		(* build template for Outer *)
		fbBuildOACData(
			bExecute		:= TRUE,
			bAddXMLHEader	:= FALSE,
			nTabIndent		:= 1,
			nOuterIndex		:= nOuterIndex,
			stOACData		:= stCACData.Outer[nOuterIndex]
		);

		(* build OAC data complete *)
		IF fbBuildOACData.bDone = TRUE THEN

			(* arrCACImage has room for OAC data and trailing </Case> tag (if required) *)
			IF SIZEOF(arrCACImage) - nCACByte - LEN('</Case>') > fbBuildOACData.nOACByte THEN

				(* add Outer data to arrCACImage *)
				(*MEMMOVE(ADR(arrCACImage[nCACByte]), ADR(fbBuildOACData.arrOACImage), fbBuildOACData.nOACByte);
				nCACByte := nCACByte + fbBuildOACData.nOACByte;*)

				nControlSize := nControlSize + fbBuildOACData.nOACByte;
				IF nControlSize <  nMaxCACImageSize  AND stCACData.NumberOfOuters <> 0 THEN
					MEMMOVE(ADR(arrCACImage[nCACByte]), ADR(fbBuildOACData.arrOACImage), fbBuildOACData.nOACByte);
					nCACByte := nCACByte + fbBuildOACData.nOACByte;
				ELSE
					bBufferOverflow	:=TRUE;
					bDone := TRUE;
					(*RETURN;*)
				END_IF


				(* last Outer in Case *)
				IF nOuterIndex = stCACData.NumberOfOuters OR  stCACData.NumberOfOuters = 0 THEN

					(* append </Case> tag *)
					strString := '</Case>';
					AppendImageData();
				END_IF
			END_IF

			eState := E_CAC_WRITEXMLIMAGE;

			(* close off fbBuildOACData *)
			fbBuildOACData(bExecute := FALSE);
		END_IF

	(* write CAC file template *)
	E_CAC_WRITEXMLIMAGE:

		(* write data to file *)
		fbWriteFile(
			sNetId		:= '',
			hFile		:= hFile,
			pWriteBuff	:= ADR(arrCACImage),
			cbWriteLen	:= nCACByte,
			bExecute	:= TRUE,
			tTimeout	:= T#1s
		);

		(* write file complete *)
		IF fbWriteFile.bBusy = FALSE THEN

			(* write file completed OK *)
			IF fbWriteFile.bError = FALSE THEN

				(* OAC required and more OAC data to be written *)
				IF nOuterIndex < stCACData.NumberOfOuters THEN

					(* re-initialise CAC byte and output image *)
					nCACByte := 0;
					nControlSize := 0;
					MEMSET(ADR(arrCACImage), 16#00, SIZEOF(arrCACImage));
					(* next Outer in Case *)
					nOuterIndex := nOuterIndex + 1;

					eState := E_CAC_BUILDXMLIMAGE;

				(* all Outers added to CAC file or Outer data not required *)
				ELSE
					eState := E_CAC_CLOSEFILE;
				END_IF
			(* write file error *)
			ELSE

				bError := TRUE;
				nErrorID := fbWriteFile.nErrID;
				eErrorState := eState;

				eState := E_CAC_CLOSEFILE;
			END_IF

			(* close off fbWriteFile *)
			fbWriteFile(bExecute := FALSE);
		END_IF


	(* close CAC template *)
	E_CAC_CLOSEFILE:

		(* close file *)
		fbCloseFile(
			sNetId		:= '',
			hFile		:= hFile,
			bExecute	:= TRUE,
			tTimeout	:= T#1s
		);

		(* close file complete *)
		IF fbCloseFile.bBusy = FALSE THEN

			(* close file completed OK and no file write error *)
			IF fbCloseFile.bError = FALSE AND bError = FALSE THEN

				eState := E_CAC_DONE;

			(* close file error or previous error with file write *)
			ELSE

				(* no previous error *)
				IF bError = FALSE THEN

					(* update error status *)
					bError := FALSE;
					nErrorID := fbCloseFile.nErrId;
					eErrorState := eState;
				END_IF

				eState := E_CAC_DONE;
			END_IF

			(* close off fbCloseFile *)
			fbCloseFile(bExecute := FALSE);
		END_IF

	(* complete *)
	E_CAC_DONE:

		bDone := TRUE;
		bBusy := FALSE;

		eState := E_CAC_IDLE;

(* unknown state *)
ELSE

	eState := E_CAC_IDLE;
END_CASE

ACTION AppendImageData:
nStringLen := LEN(strString);
nControlSize := nControlSize + nStringLen;
IF nControlSize <  nMaxCACImageSize THEN
	MEMMOVE(ADR(arrCACImage[nCACByte]), ADR(strString), nStringLen);
	nCACByte := nCACByte + nStringLen;
ELSE
	bBufferOverflow	:=TRUE;
	bDone := TRUE;
	(*RETURN;*)
END_IF
END_ACTION

END_FUNCTION_BLOCK

// ---- POUs/_Exclude/FB_CHM_ClearArchive.TcPOU
(* scans CHM archive and deletes files and folders older than tMaxArchiveAge *)
FUNCTION_BLOCK FB_CHM_ClearArchive
VAR_INPUT
	bExecute				: BOOL;			(* set TRUE to scan archive for old folders and files *)
	tMaxArchiveAge		: TIME;			(* max file age, older files/folders will be deleted *)
	strLocalCHMPath		: STRING(255);	(* CaseTrace CHM folder path *)
	sSystemTime			: TIMESTRUCT;	(* current system time *)
END_VAR
VAR_OUTPUT
	bDone				: BOOL;			(* TRUE = scan complete *)
	bBusy				: BOOL;			(* TRUE = scan in progress *)
	bError				: BOOL;			(* TRUE = scan error *)
	nErrorID				: UDINT;		(* error code *)
	nFoldersDeleted		: UDINT;		(* total folders deleted *)
	nCHMFilesDeleted		: UDINT;		(* total CHM files deleted *)
END_VAR
VAR
	fbExecute				: R_TRIG;
	eState				: E_CHM_State;
	eErrorState			: E_CHM_State;
	nSourceAge			: T_ULARGE_INTEGER;
	nFoldersFound			: UDINT;
	nCHMFilesFound		: UDINT;

	fbFindFolder			: FB_EnumFindFileEntry;
	eFolderCmd 			: E_EnumCmdType := eEnumCmd_First;
	strFolder				: STRING(255);

	fbFindFile				: FB_EnumFindFileEntry;
	eFileCmd 				: E_EnumCmdType := eEnumCmd_First;
	strFileName			: STRING(255);

	fbDeleteFile			: FB_FileDelete;
	fbDeleteFolder			: FB_RemoveDir;
END_VAR

fbExecute(CLK := bExecute);

CASE eState OF

	(* idle *)
	E_CHM_IDLE:

		(* rising edge of bExecute *)
		IF fbExecute.Q = TRUE THEN

			(* update outputs *)
			bDone := FALSE;
			bBusy := TRUE;
			bError := FALSE;
			nErrorID := 0;

			(* reset values *)
			nFoldersDeleted := 0;
			nCHMFilesDeleted := 0;
			nFoldersFound := 0;
			nCHMFilesFound := 0;

			strFolder := '';
			eFolderCmd := eEnumCmd_First;
			strFileName := '';
			eFileCmd := eEnumCmd_First;

			eState := E_CHM_FINDFOLDER;

		(* bExecute has been reset *)
		ELSIF bExecute = FALSE THEN

			(* reset outputs *)
			bDone := FALSE;
			bBusy := FALSE;
			bError := FALSE;
			nErrorID := 0;
		END_IF


	(* date folders *)
	E_CHM_FINDFOLDER:

		(* get list of date folders in "..CaseTrace\CHM\Archive\" *)
		fbFindFolder(
			sNetId		:= '',
			sPathName	:= CONCAT(strLocalCHMPath, 'Archive\*.'),
			eCmd		:= eFolderCmd,
			bExecute	:= TRUE,
			tTimeout	:= T#5s
		);

		(* find folder complete *)
		IF fbFindFolder.bBusy = FALSE THEN

			(* find folder completed OK *)
			IF fbFindFolder.bError = FALSE THEN

				(* file list complete *)
				IF fbFindFolder.bEOE = TRUE THEN

					eFolderCmd := eEnumCmd_First;

					eState := E_CHM_DONE;

				(* file found *)
				ELSE

					(* first 2 folders are '.' and '..' *)
					IF fbFindFolder.stFindFile.sFileName = '.' OR fbFindFolder.stFindFile.sFileName = '..' THEN

						(* next file *)
						eFolderCmd := eEnumCmd_Next;

					(* folder found *)
					ELSE

						(* update counter *)
						nFoldersFound := nFoldersFound + 1;

						(* FolderAge = SystemTime - FileTime *)
						nSourceAge := UInt64Sub64(F_FileTimeToULarge(SYSTEMTIME_TO_FILETIME(sSystemTime)), F_FileTimeToULarge(fbFindFolder.stFindFile.creationTime));

						(* folder is older than max age (converted to 64-bit format) *)
						IF UInt64Cmp64(nSourceAge, UInt32x32To64(TIME_TO_UDINT(tMaxArchiveAge), 10000)) = 1 THEN

							(* folder found *)
							strFolder := fbFindFolder.stFindFile.sFileName;

							eState := E_CHM_FINDFILE;
						END_IF

						(* next folder on next pass *)
						eFolderCmd := eEnumCmd_Next;
					END_IF
				END_IF

			(* find folder error *)
			ELSE

				(* update outputs *)
				bError := TRUE;
				nErrorID := fbFindFolder.nErrID;
				eErrorState := eState;

				eFolderCmd := eEnumCmd_First;

				eState := E_CHM_DONE;
			END_IF

			(* close off fbFindFolder *)
			fbFindFolder(bExecute := FALSE);
		END_IF


	(* find files in folder *)
	E_CHM_FINDFILE:

		(* get list of files *)
		fbFindFile(
			sNetId		:= '',
			sPathName	:= F_CONCAT4(strLocalCHMPath, 'Archive\', strFolder, '\*.*'),
			eCmd		:= eFileCmd,
			bExecute	:= TRUE,
			tTimeout	:= T#5s
		);

		(* find date complete *)
		IF fbFindFile.bBusy = FALSE THEN

			(* find file completed OK *)
			IF fbFindFile.bError = FALSE THEN

				(* file list complete *)
				IF fbFindFile.bEOE = TRUE THEN

					eFileCmd := eEnumCmd_First;

					eState := E_CHM_DELETEFOLDER;

				(* file found *)
				ELSE

					(* first 2 files could be '.' and '..' *)
					IF fbFindFile.stFindFile.sFileName = '.' OR fbFindFile.stFindFile.sFileName = '..' THEN

						(* next file *)
						eFileCmd := eEnumCmd_Next;

					(* folder found *)
					ELSE

						(* count files in folder *)
						nCHMFilesFound := nCHMFilesFound + 1;
	
						(* FileAge = SystemTime - FileTime *)
						nSourceAge := UInt64Sub64(F_FileTimeToULarge(SYSTEMTIME_TO_FILETIME(sSystemTime)), F_FileTimeToULarge(fbFindFile.stFindFile.creationTime));

						(* source file is older than max age (converted to 64-bit format) *)
						IF UInt64Cmp64(nSourceAge, UInt32x32To64(TIME_TO_UDINT(tMaxArchiveAge), 10000)) = 1 THEN
	
							(* date folder found *)
							strFileName := fbFindFile.stFindFile.sFileName;
	
							eState := E_CHM_DELETEFILE;
						END_IF
	
						(* next folder *)
						eFileCmd := eEnumCmd_Next;
					END_IF
				END_IF

			(* find file error *)
			ELSE

				(* update outputs *)
				bError := TRUE;
				nErrorID := fbFindFile.nErrID;
				eErrorState := eState;

				eFileCmd := eEnumCmd_First;

				eState := E_CHM_FINDFOLDER;
			END_IF

			(* close off fbFindFile *)
			fbFindFile(bExecute := FALSE);
		END_IF


	(* delete old file *)
	E_CHM_DELETEFILE:

		(* delete files *)
		fbDeleteFile(
			sNetId		:= '',
			sPathName	:= F_CONCAT5(strLocalCHMPath, 'Archive\', strFolder, '\', strFileName),
			ePath		:= PATH_GENERIC,
			bExecute	:= TRUE,
			tTimeout	:= T#1s
		);

		(* delete file complete *)
		IF fbDeleteFile.bBusy = FALSE THEN

			(* delete file completed OK *)
			IF fbDeleteFile.bError = FALSE THEN

				(* count files deleted from current folder *)
				nCHMFilesDeleted := nCHMFilesDeleted + 1;
			END_IF

			eState := E_CHM_FINDFILE;

			(* close off fbDeleteFile *)
			fbDeleteFile(bExecute := FALSE);
		END_IF


	(* delete old folder *)
	E_CHM_DELETEFOLDER:

		(* delete folder *)
		fbDeleteFolder(
			sNetId		:= '',
			sPathName	:= F_CONCAT3(strLocalCHMPath, 'Archive\', strFolder),
			ePath		:= PATH_GENERIC,
			bExecute	:= TRUE,
			tTimeout	:= T#1s
		);

		(* delete folder complete *)
		IF fbDeleteFolder.bBusy = FALSE THEN

			(* delete folder complete *)
			IF fbDeleteFolder.bError = FALSE THEN

				(* count folder deleted *)
				nFoldersDeleted := nFoldersDeleted + 1;
			END_IF

			eState := E_CHM_FINDFOLDER;

			(* close off fbDeleteFolder *)
			fbDeleteFolder(bExecute := FALSE);
		END_IF


	(* complete *)
	E_CHM_DONE:

		(* update outputs *)
		bBusy := FALSE;
		bDone := TRUE;

		eState := E_CHM_IDLE;


(* unknown state *)
ELSE

	eState := E_CHM_IDLE;

	bDone := FALSE;
	bBusy := FALSE;
	bError := FALSE;
	nErrorID := 0;
END_CASE

END_FUNCTION_BLOCK

// ---- POUs/_Exclude/FB_CX_NVData_NOVRAM_4K.TcPOU
(* stores data in local NOV/DP-RAM device (CX only) *)
FUNCTION_BLOCK FB_CX_NVData_NOVRAM_4K
VAR_INPUT
	bEnable				: BOOL;				(* set TRUE to enable NOVRAM data storage *)
	bExport				: BOOL;				(* set TRUE to export data to XML file, format is compatible with TSM export file *)
	bImport				: BOOL;				(* set TRUE to import data from XML file, format is compatible with TSM export file *)
	pCtrlData			: POINTER TO WORD;	(* pointer to 1st byte of ctrl data to be stored *)
	nCtrlBytes			: UDINT;			(* no of ctrl data bytes to be stored *)
	strTransferPathFile	: T_MaxString;		(* transfer file name for export/import *)
END_VAR
VAR_OUTPUT
	bNVDataInitOK		: BOOL;				(* TRUE = initialisation completed OK *)
	bError				: BOOL;				(* TRUE = initialisation error (device or checksum) *)
	nUpdates			: UDINT;			(* number of NOVRAM writes completed *)
	nDeviceID			: WORD;				(* NOVRAM device ID *)
END_VAR
VAR
	eState				: E_CX_NVDataCtrlState;
	eErrorState			: E_CX_NVDataCtrlState;
	arrInputData		: ARRAY[0..4095] OF BYTE;
	arrOutputData		: ARRAY[0..4095] OF BYTE;

	fbExport			: R_TRIG;
	bExportReq			: BOOL;
	fbImport			: R_TRIG;
	bImportReq			: BOOL;

	fbTaskTime			: FB_SYSTEM_TaskInfo;
	nNVReadBlockSize	: UDINT;
	nNVWriteBlockSize	: UDINT;
	nChecksumBlockSize	: UDINT;
	pNVData				: POINTER TO BYTE;

	fbGetCXPlatform		: FB_CxGetDeviceIdentificationEx;
	nMaxDataBytes		: UDINT;
	fbGetDeviceID		: FB_CX_GetDeviceID;
	fbGetDeviceInfo		: FB_GetDPRAMInfo;
	sDeviceInfo			: ST_NovRamAddrInfo;

	nActiveDataArea		: UINT;
	pChecksum			: POINTER TO WORD;
	nCalcChecksum		: WORD;
	nNVBlockOffset		: UDINT;
	nNVBlockBytes		: UDINT;
	nIndexOffset		: UDINT;
	nIndexBlockBytes	: UDINT;
	fbTransferData		: FB_CX_NVData_Transfer;
END_VAR
(*
-------------------------------------------------------------------------------------------------
Date		Version	Author	Comments
-------------------------------------------------------------------------------------------------
30/01/2015	3.00.00	PB		Initial release

-------------------------------------------------------------------------------------------------

*)

(* rising edge of bExport *)
fbExport(CLK := bExport);
IF fbExport.Q = TRUE THEN

	(* set flag to export data at next opportunity *)
	bExportReq := TRUE;
END_IF

(* rising edge of bImport *)
fbImport(CLK := bImport);
IF fbImport.Q = TRUE THEN

	(* set flag to import data at next opportunity *)
	bImportReq := TRUE;
END_IF


CASE eState OF

	(* IDLE state *)
	E_CX_NVDATA_IDLE:

		(* NOVRAM storage is enabled *)
		IF bEnable = TRUE THEN

			(* get current task time *)
			fbTaskTime();

			(* initialise vars *)
			nActiveDataArea := 0;
			nMaxDataBytes := SIZEOF(arrInputData);
			MEMSET(ADR(sDeviceInfo), 16#00, SIZEOF(sDeviceInfo));

			(* initialise outputs *)
			nUpdates := 0;
			nDeviceID := 0;

			eState := E_CX_NVDATA_PLATFORM;

		(* else *)
		ELSE

			bNVDataInitOK := FALSE;
			bError := FALSE;
		END_IF


	(* find CX type *)
	E_CX_NVDATA_PLATFORM:

		(* get CX platform type *)
		fbGetCXPlatform(
			bExecute	:= TRUE,
			tTimeout	:= T#1s
		);

		(* get CX platform type complete *)
		IF fbGetCXPlatform.bBusy = FALSE THEN

			(* get CX platform type completed OK *)
			IF fbGetCXPlatform.bError = FALSE THEN

				(* Block sizes have been selected to use approx 5% resource in 1ms PLC task on CX1020 and CX2020. *)
				(* Processor resource should be lower on CX1030 and CX2030/CX2040 due to higher processor speed. *)
				(* FB will be adjusted for other platforms when they are available for testing *)

				(* CX1020/CX1030 platform *)
				IF FIND(fbGetCXPlatform.stDevIdent.strHardwareModel, '1020') > 0 OR FIND(fbGetCXPlatform.stDevIdent.strHardwareModel, '1030') > 0 THEN

					(* NOVRAM block access size per 1ms of PLC cycle time:  READ = 32 bytes/ms, WRITE = 128 bytes/ms *)
					nNVReadBlockSize := MIN(LREAL_TO_UDINT(fbTaskTime.fTaskTimeMicrosecs * 32.0 / 1000.0), 32);
					nNVWriteBlockSize := MIN(LREAL_TO_UDINT(fbTaskTime.fTaskTimeMicrosecs * 128.0 / 1000.0), 128);

					(* checksum block size:  512 bytes/ms PLC task time *)
					nChecksumBlockSize := LREAL_TO_UDINT(fbTaskTime.fTaskTimeMicrosecs * 512.0 / 1000.0);

				(* CX2020/CX2030/CX2040 platform *)
				ELSIF FIND(fbGetCXPlatform.stDevIdent.strHardwareModel, '2020') > 0 OR FIND(fbGetCXPlatform.stDevIdent.strHardwareModel, '2030') > 0 OR FIND(fbGetCXPlatform.stDevIdent.strHardwareModel, '2040') > 0 THEN

					(* NOVRAM block access size per 1ms of PLC cycle time:  READ = 64 bytes/ms, WRITE = 1024 bytes/ms *)
					nNVReadBlockSize := MIN(LREAL_TO_UINT(fbTaskTime.fTaskTimeMicrosecs * 64.0 / 1000.0), 64);
					nNVWriteBlockSize := MIN(LREAL_TO_UINT(fbTaskTime.fTaskTimeMicrosecs * 1024.0 / 1000.0), 1024);

					(* checksum block size per 1ms of PLC cycle time:  1024 bytes/ms *)
					nChecksumBlockSize := LREAL_TO_UINT(fbTaskTime.fTaskTimeMicrosecs * 1024.0 / 1000.0);

				(* CX2020/CX2030/CX2040 platform *)
				ELSIF FIND(fbGetCXPlatform.stDevIdent.strTargetType, 'PC') > 0  THEN

					(* NOVRAM block access size per 1ms of PLC cycle time:  READ = 64 bytes/ms, WRITE = 1024 bytes/ms *)
					nNVReadBlockSize := MIN(LREAL_TO_UINT(fbTaskTime.fTaskTimeMicrosecs * 64.0 / 1000.0), 64);
					nNVWriteBlockSize := MIN(LREAL_TO_UINT(fbTaskTime.fTaskTimeMicrosecs * 1024.0 / 1000.0), 1024);

					(* checksum block size per 1ms of PLC cycle time:  1024 bytes/ms *)
					nChecksumBlockSize := LREAL_TO_UINT(fbTaskTime.fTaskTimeMicrosecs * 1024.0 / 1000.0);
				END_IF

				(* DeviceID is not specified *)
				IF nDeviceID = 0 THEN

					(* search CX for NOVRAM device *)
					eState := E_CX_NVDATA_DEVICEID;

				(* DeviceID is specifeid *)
				ELSE

					(* use specified DeviceID *)
					eState := E_CX_NVDATA_DEVICEINFO;
				END_IF

			(* get CX platform type error *)
			ELSE

				bError := TRUE;
				eErrorState := eState;

				eState := E_CX_NVDATA_DONE;
			END_IF

			(* cloes off fbGetCXPlatform *)
			fbGetCXPlatform(bExecute := FALSE);
		END_IF


	(* find NOVRAM device ID *)
	E_CX_NVDATA_DEVICEID:

		(* get DeviceID for DPRAM *)
		fbGetDeviceID(
			bExecute	:= TRUE,
			eDeviceType	:= IODEVICETYPE_DPRAM
		);

		(* get DeviceID complete *)
		IF fbGetDeviceID.bDone = TRUE THEN

			(* get DeviceID completed OK and NOVRAM device found *)
			IF fbGetDeviceID.bDone = TRUE AND fbGetDeviceID.bDeviceFound = TRUE THEN

				(* DeviceID of NOVRAM device *)
				nDeviceID := fbGetDeviceID.nDeviceID;

				eState := E_CX_NVDATA_DEVICEINFO;

			(* fbGetDeviceID error of NOVRAM device not found *)
			ELSE

				(* reset nDeviceID *)
				nDeviceID := 0;

				(* update error status *)
				bError := TRUE;
				eErrorState := eState;

				eState := E_CX_NVDATA_DONE;
			END_IF

			(* close off fbGetDeviceID *)
			fbGetDeviceID(bExecute := FALSE);
		END_IF


	(* read info of NOVRAM device *)
	E_CX_NVDATA_DEVICEINFO:

		(* get device info *)
		fbGetDeviceInfo(
			nDevId	:= nDeviceID,
			bExecute:= TRUE,
			tTimeOut:= T#1s
		);

		(* device info read complete *)
		IF fbGetDeviceInfo.bBusy = FALSE THEN

			(* NOVRAM info read successful *)
			IF fbGetDeviceInfo.bError = FALSE THEN

				(* set up config data for NV data block *)
				sDeviceInfo := fbGetDeviceInfo.stInfo;

				(* maximum number of NV bytes that can be handled *)
				nMaxDataBytes := sDeviceInfo.iCardMemSize / 2;

				(* specified number of data bytes is valid *)
				IF nCtrlBytes <= nMaxDataBytes THEN

					(* read primary data from NOVRAM *)
					nActiveDataArea := 1;
					pNVData := sDeviceInfo.pCardAddress;

					(* initial byte offset and block size for 1st scan *)
					nNVBlockOffset := 0;
					nNVBlockBytes := MIN(nNVReadBlockSize, nCtrlBytes - nNVBlockOffset);

					eState := E_CX_NVDATA_READ;

				(* memory area too large *)
				ELSE

					bError := TRUE;
					eErrorState := eState;
	
					eState := E_CX_NVDATA_DONE;
				END_IF

			(* unable to read NOVRAM info *)
			ELSE

				bError := TRUE;
				eErrorState := eState;

				eState := E_CX_NVDATA_DONE;
			END_IF

			(* close fbGetDeviceInfo *)
			fbGetDeviceInfo(bExecute:= FALSE);
		END_IF


	(* read data to NOVRAM *)
	E_CX_NVDATA_READ:

		(* restore NOVRAM data into arrInputData in blocks *)
		MEMMOVE(ADR(arrInputData[nNVBlockOffset]), F_PointerToByteADD(pNVData, nNVBlockOffset), nNVBlockBytes);

		(* update memory offset values *)
		nNVBlockOffset := nNVBlockOffset + nNVBlockBytes;
		nNVBlockBytes := MIN(nNVReadBlockSize, nCtrlBytes - nNVBlockOffset);

		(* all bytes transferred *)
		IF nNVBlockOffset >= nCtrlBytes THEN

			(* initialise checksum block vars *)
			nIndexOffset := 0;
			nIndexBlockBytes := MIN(nChecksumBlockSize, nCtrlBytes - 2 - nIndexOffset);
			nCalcChecksum := 16#FFFF;

			eState := E_CX_NVDATA_VALIDATE;
		END_IF


	(* verify checksum *)
	E_CX_NVDATA_VALIDATE:

		(* calculate checksum on block of data *)
		nCalcChecksum := F_DATA_TO_CRC16_CCITT(ADR(arrInputData[nIndexOffset]), nIndexBlockBytes, nCalcChecksum);

		(* update nIndexOffset and nIndexBlockBytes for next pass *)
		nIndexOffset := nIndexOffset + nIndexBlockBytes;
		nIndexBlockBytes := MIN(nChecksumBlockSize, nCtrlBytes - 2 - nIndexOffset);

		(* checksum completed for all bytes *)
		IF nIndexOffset >= nCtrlBytes - 2 THEN

			(* pointer to restored checksum in arrInputData *)
			pChecksum := ADR(arrInputData[nCtrlBytes - 2]);

			(* calculated checksum = restored checksum *)
			IF nCalcChecksum = pChecksum^ THEN

				(* restore NOVRAM data into snapshot array *)
				MEMMOVE(pCtrlData, ADR(arrInputData), nCtrlBytes);
				bNVDataInitOK := TRUE;

				eState := E_CX_NVDATA_COMPARE;

			(* calculated checksum <> restored checksum *)
			ELSE

				(* primary data failed *)
				IF nActiveDataArea = 1 THEN

					(* move to secondary data *)
					nActiveDataArea := 2;

					(* calculate pointers needed to restore secondary data *)
					pNVData := F_PointerToByteADD(pNVData, sDeviceInfo.iCardMemSize / 2);

					(* initial byte offset and block size for 1st scan *)
					nNVBlockOffset := 0;
					nNVBlockBytes := MIN(nNVWriteBlockSize, nCtrlBytes - nNVBlockOffset);

					eState := E_CX_NVDATA_READ;

				(* secondary data failed *)
				ELSE

					(* checksum invalid for primary and secondary data, clear arrInput data *)
					MEMSET(ADR(arrInputData), 16#00, SIZEOF(arrInputData));
					bError := TRUE;
					eErrorState := eState;
					(* data will be written to NOVRAM on COMPARE cycle, unless all values are 0 when no update will occur *)

					eState := E_CX_NVDATA_COMPARE;
				END_IF
			END_IF
		END_IF


	(* snapshot data *)
	E_CX_NVDATA_COMPARE:

		(* FB is enabled *)
		IF bEnable = TRUE THEN

			(* specified number of data bytes is valid *)
			IF nCtrlBytes <= nMaxDataBytes THEN

				(* export data requested *)
				IF bExportReq = TRUE THEN

					(* cancel export flag *)
					bExportReq := FALSE;

					eState := E_CX_NVDATA_EXPORT;

				(* import data requested *)
				ELSIF bImportReq = TRUE THEN

					(* cancel import flag *)
					bImportReq := FALSE;

					eState := E_CX_NVDATA_IMPORT;

				(* check for change of data *)
				ELSE

					(* snapshot data into arrOutputData *)
					MEMMOVE(ADR(arrOutputData), pCtrlData, nCtrlBytes - 2);

					(* snapshot data block does not match terminal data block *)
					IF MEMCMP(ADR(arrOutputData), ADR(arrInputData), nCtrlBytes - 2) <> 0 THEN

						(* initialise checksum block vars *)
						nIndexOffset := 0;
						nIndexBlockBytes := MIN(nChecksumBlockSize, nCtrlBytes - 2 - nIndexOffset);
						nCalcChecksum := 16#FFFF;

						eState := E_CX_NVDATA_CHECKSUM;
					END_IF
				END_IF

			(* memory area too large *)
			ELSE

				bError := TRUE;
				eErrorState := eState;

				eState := E_CX_NVDATA_DONE;
			END_IF

		(* FB is disabled *)
		ELSE

			eState := E_CX_NVDATA_DONE;
		END_IF


	(* calculate checksum for output data *)
	E_CX_NVDATA_CHECKSUM:

		(* calculate checksum on block of data *)
		nCalcChecksum := F_DATA_TO_CRC16_CCITT(ADR(arrOutputData[nIndexOffset]), nIndexBlockBytes, nCalcChecksum);

		(* update nIndexOffset and nIndexBlockBytes for next pass *)
		nIndexOffset := nIndexOffset + nIndexBlockBytes;
		nIndexBlockBytes := MIN(nChecksumBlockSize, nCtrlBytes - 2 - nIndexOffset);

		(* checksum completed for all bytes *)
		IF nIndexOffset >= nCtrlBytes - 2 THEN

			(* pointer to restored checksum in arrInputData *)
			pChecksum := ADR(arrOutputData[nCtrlBytes - 2]);
			pChecksum^ := nCalcChecksum;

			(* write primary data from NOVRAM *)
			nActiveDataArea := 1;
			pNVData := sDeviceInfo.pCardAddress;

			(* initial byte offset and block size for 1st scan *)
			nNVBlockOffset := 0;
			nNVBlockBytes := MIN(nNVWriteBlockSize, nCtrlBytes - nNVBlockOffset);

			eState := E_CX_NVDATA_WRITE;
		END_IF


	(* write data *)
	E_CX_NVDATA_WRITE:

		(* move arrOutputData to NOVRAM *)
		MEMMOVE(F_PointerToByteADD(pNVData, nNVBlockOffset), ADR(arrOutputData[nNVBlockOffset]), nNVBlockBytes);

		(* update memory offset values *)
		nNVBlockOffset := nNVBlockOffset + nNVBlockBytes;
		nNVBlockBytes := MIN(nNVWriteBlockSize, nCtrlBytes - nNVBlockOffset);

		(* all bytes transferred *)
		IF nNVBlockOffset >= nCtrlBytes THEN

			(* primary data written *)
			IF nActiveDataArea = 1 THEN

				(* write primary data from NOVRAM *)
				nActiveDataArea := 2;
				pNVData := F_PointerToByteADD(sDeviceInfo.pCardAddress, sDeviceInfo.iCardMemSize / 2);

				(* initial byte offset and block size for 1st scan *)
				nNVBlockOffset := 0;
				nNVBlockBytes := MIN(nNVWriteBlockSize, nCtrlBytes - nNVBlockOffset);

			(* secondary data complete *)
			ELSE

				(* update outputs *)
				bNVDataInitOK := TRUE;
				bError := FALSE;
				nActiveDataArea := 0;
				nUpdates := nUpdates + 1;

				(* copy arrOutputData to arrInputData *)
				MEMMOVE(ADR(arrInputData), ADR(arrOutputData), nCtrlBytes);

				(* update checksum in pCtrlData area *)
				pChecksum := F_PointerToWordADD(pCtrlData, nCtrlBytes - 2);
				pChecksum^ := nCalcChecksum;

				eState := E_CX_NVDATA_COMPARE;
			END_IF
		END_IF


	(* export data to XML file *)
	E_CX_NVDATA_EXPORT:

		(* export data from arrInputData to XML file *)
		fbTransferData(
			bExecute		:= TRUE,
			bImport			:= FALSE,
			nMaxBlockSize	:= nChecksumBlockSize / 2,
			pCtrlData		:= ADR(arrInputData),
			nCtrlBytes		:= nCtrlBytes,
			strPathFile		:= strTransferPathFile
		);

		(* export data complete *)
		IF fbTransferData.bDone = TRUE THEN

			eState := E_CX_NVDATA_COMPARE;

			(* close off fbTransferData *)
			fbTransferData(bExecute := FALSE);
		END_IF


	(* import data to XML file *)
	E_CX_NVDATA_IMPORT:

		(* import data from XML file to arrOutputData *)
		fbTransferData(
			bExecute		:= TRUE,
			bImport			:= TRUE,
			nMaxBlockSize	:= nChecksumBlockSize / 2,
			pCtrlData		:= ADR(arrOutputData),
			nCtrlBytes		:= SIZEOF(arrOutputData),
			strPathFile		:= strTransferPathFile
		);

		(* import data complete *)
		IF fbTransferData.bDone = TRUE THEN

			(* import data completed OK *)
			IF fbTransferData.bError = FALSE THEN

				(* move data loaded to pCtrlData *)
				MEMMOVE(pCtrlData, ADR(arrOutputData), fbTransferData.nTotalDataBytes);

				eState := E_CX_NVDATA_COMPARE;

			(* import data error *)
			ELSE

				eState := E_CX_NVDATA_COMPARE;
			END_IF

			(* close off fbTransferData *)
			fbTransferData(bExecute := FALSE);
		END_IF


	(* access complete *)
	E_CX_NVDATA_DONE:

		;

END_CASE

END_FUNCTION_BLOCK

// ---- POUs/_Exclude/FB_MemoryMonitor_32K.TcPOU
(* monitor memory area for change of data, max 64Kbytes *)
FUNCTION_BLOCK FB_MemoryMonitor_32K
VAR_INPUT
	bEnable			: BOOL;		(* set TRUE to enable monitoring *)
	pSourceData		: POINTER TO BYTE;	(* pointer to source data *)
	nSourceBytes	: UDINT;	(* no of data bytes *)
	tUpdateTime		: TIME;		(* update time *)
END_VAR
VAR_OUTPUT
	bDataChanged	: BOOL;		(* TRUE = data changed *)
	nTotalChanges	: UDINT;	(* total number of memory changes detected *)
END_VAR
VAR
	arrData			: ARRAY[0..32767] OF BYTE;
	fbUpdateTimer	: FB_PulseGenerator;
END_VAR
(*
-------------------------------------------------------------------------------------------------
Date		Version	Author	Comments
-------------------------------------------------------------------------------------------------
30/01/2015	3.00.00	PB		Initial release

-------------------------------------------------------------------------------------------------
*)

(* update timer *)
fbUpdateTimer(
	bEnable		:= bEnable,
	tPeriod		:= tUpdateTime
);

(* data not changed on last pass *)
IF bDataChanged = FALSE THEN

	(* check for change of data *)
	IF fbUpdateTimer.bOutput = TRUE THEN

		(* source data in array has changed *)
		IF MEMCMP(pSourceData, ADR(arrData), nSourceBytes) <> 0 THEN

			nTotalChanges := nTotalChanges + 1;
			bDataChanged := TRUE;
		END_IF
	END_IF

(* data change detected on last pass *)
ELSE

	(* move data from source to target *)
	MEMMOVE(ADR(arrData), pSourceData, nSourceBytes);
	bDataChanged := FALSE;
END_IF

END_FUNCTION_BLOCK

// ---- POUs/_Exclude/FB_MemoryMonitor_4K.TcPOU
(* monitor memory area for change of data, max 4Kbytes *)
FUNCTION_BLOCK FB_MemoryMonitor_4K
VAR_INPUT
	bEnable			: BOOL;		(* set TRUE to enable monitoring *)
	pSourceData		: POINTER TO BYTE;	(* pointer to source data *)
	nSourceBytes	: UDINT;	(* no of data bytes *)
	tUpdateTime		: TIME;		(* update time *)
END_VAR
VAR_OUTPUT
	bDataChanged	: BOOL;		(* TRUE = data changed *)
	nTotalChanges	: UDINT;	(* total number of memory changes detected *)
END_VAR
VAR
	arrData			: ARRAY[0..4095] OF BYTE;
	fbUpdateTimer	: FB_PulseGenerator;
END_VAR
(*
-------------------------------------------------------------------------------------------------
Date		Version	Author	Comments
-------------------------------------------------------------------------------------------------
30/01/2015	3.00.00	PB		Initial release

-------------------------------------------------------------------------------------------------
*)

(* update timer *)
fbUpdateTimer(
	bEnable		:= bEnable,
	tPeriod		:= tUpdateTime
);

(* data not changed on last pass *)
IF bDataChanged = FALSE THEN

	(* check for change of data *)
	IF fbUpdateTimer.bOutput = TRUE THEN

		(* source data in array has changed *)
		IF MEMCMP(pSourceData, ADR(arrData), nSourceBytes) <> 0 THEN

			nTotalChanges := nTotalChanges + 1;
			bDataChanged := TRUE;
		END_IF
	END_IF

(* data change detected on last pass *)
ELSE

	(* move data from source to target *)
	MEMMOVE(ADR(arrData), pSourceData, nSourceBytes);
	bDataChanged := FALSE;
END_IF

END_FUNCTION_BLOCK

// ---- POUs/_Exclude/FB_OUTER_CompleteDataFromConfirmation.TcPOU
 FUNCTION_BLOCK FB_OUTER_CompleteDataFromConfirmation
VAR_INPUT
	bExecute								: BOOL;		(* set TRUE to scan arrOuterStatus for completed Outers *)
	bValidationTimeout					: BOOL;
	(*bOuterCameraDone					: BOOL;*)
	(*bConfirmationCameraDone			: BOOL;*)
(*	stOuterValidationCameraLastCodes	: ST_SCANNER_ImageData;*)
	stBarcodeConfirmationCameraLastCodes	: ST_SCANNER_ImageData;
	(*nPackPos1								: INT 	:=1;
	nPackPos2								: INT	:=2;*)
	bUseInterimCodeForValidation		: BOOL;
	sLocalOCVPath							: STRING(255);
	stCTDateTime							: ST_SYSTEM_DateTime;	(* CaseTrace date/time structure *)
	bQAReject								: BOOL;
END_VAR
VAR_IN_OUT
	stProductInstruction		: ST_PCM_Status;					(* Product Instruction *)
	stOuterRejectReasons		: ST_RejectReasonsForOuter;
	aOuterStatus				: ARRAY[1..cMAX_OUTER_STATUS_QUEUE] OF ST_OUTER_Status;	(* Outer status register *)
	aOCVPackStatus			: ARRAY[1..cMAX_OUTER_STATUS_QUEUE] OF ST_OUTER_Status;	(* Outer status register *)
	stOuterStatusHMI			: ST_HMI_OuterStatus;
END_VAR
VAR_OUTPUT
	bDone						: BOOL;			(* TRUE = validation complete *)
	bBusy						: BOOL;			(* TRUE = validation in progress *)

	stLastOuterStatus			: ST_OUTER_Status;

	sLastReadOuterBarcode	: T_OUTER_Barcode;
	sLastReadConfPackCode1	: T_PACK_Barcode;
	(*sLastReadConfPackCode2 	: T_PACK_Barcode;*)
	(*aConfPackCodeInPosition		: ARRAY[0..1] OF T_PACK_Barcode;*)
	sOCVRejectCode			: T_RejectCode;
	nOCVRejectID				: UINT;
	bPackDataFoundInStruct	: BOOL;
	nInhibitOCVRestore		: BOOL;
	bReadyToOCVResotre		: BOOL;
	nOutersCompleted			: UDINT;

END_VAR
VAR
	eState						: E_OUTER_AgrregationState;
	fbExecute					: R_TRIG;
	fbTimeOut					: R_TRIG;
	stSystemTime				: TIMESTRUCT;

	(*nAggregartionPackCode	: INT;*)

	nOuterIndex				: INT;
	(*nMaxOuterIndex				: INT;*)
	nPackIndex				: INT;

	aOCVFileCodeName		: ARRAY[1..2] OF T_MaxString;
	bReffedOCVExec			: BOOL;
	fbOCVRefeed				: FB_OUTER_RefeedOCVFilesWtihError; (*FB_PACK_RefeedOCVFilesWtihError;*)

	stPacksDataFromOCV1	: ST_OUTER_Status;
	stPacksDataFromOCV2	: ST_OUTER_Status;

	nTrigID						: UDINT;
	(*aLogTrigID					: ARRAY[0..5] OF UDINT;*)
	nNewOuterTrigID			: UDINT;

	(*aPackStatusValue				: ARRAY[0..10] OF INT;
	aRejectCodePointer            		: ARRAY[0..10] OF STRING(10);

	fbValidatePack					: FB_CODE_ValidateExplicitCode;*)

	nErrorCounter1			: INT;
	nErrorCounter2			: INT;
	nErrorCounter3			: INT;

	tonTestTimer				: TON;
	aLogTimer 					: ARRAY[0..100] OF TIME;
END_VAR

fbExecute(CLK := bExecute);
fbTimeOut(CLK := bValidationTimeout);

stSystemTime := stCTDateTime.sSystemTime;

tonTestTimer(In:= bBusy AND NOT bDone, PT:= t#5000ms);
IF fbTimeOut.Q THEN

		aOuterStatus[1].stOACData.ProductionDate := F_StringWildcard('#YYYYMMDD#', stSystemTime);
		aOuterStatus[1].stOACData.ProductionTime := F_StringWildcard('#hhmmss#', stSystemTime);
		aOuterStatus[1].stOACData.ProductionTimeOffset := F_SYSTEM_SystemTimeOffsetToHHMM(stCTDateTime.nSystemTimeOffset);

		aOuterStatus[1].stOACData.OuterTimeStamp :=F_SYSTEM_SystemTimeAsISO8601(stCTDateTime.sSystemTime, stCTDateTime.sUTCTimeZoneOffset );
		aOuterStatus[1].stOACData.RetailSKU := stProductInstruction.sRetailSKU;
		aOuterStatus[1].stOACData.OuterMachine.ProductionSite :=  stProductInstruction.sProductionSite;
		aOuterStatus[1].stOACData.OuterMachine.ProductionLine := stProductInstruction.sProductionLine;
		aOuterStatus[1].stOACData.BatchNumber := stProductInstruction.sBatchNumber;
		aOuterStatus[1].stOACData.CodingAndTrackingMode := stProductInstruction.nOpMode;

		aOuterStatus[1].stOACData.AcceptanceLevel := stProductInstruction.nAcceptanceLevel;
		aOuterStatus[1].stOACData.NumberOfPacks	:= stProductInstruction.nPacksPerOuter;

		(*IF  NOT bConfirmationCameraDone	THEN
			aOuterStatus[1].sDataSourceTracker	:= 'T_OUT_PCC';
		ELSE
			aOuterStatus[1].sDataSourceTracker	:= 'T_OUT_FB';
		END_IF*)
		aOuterStatus[1].sDataSourceTracker	:= 'T_OUT_FB';

		aOuterStatus[1].nStatus.9 := TRUE;
		aOuterStatus[1].nTriggerID := nNewOuterTrigID;
		aOuterStatus[1].stOACData.OuterRejectCode := stOuterRejectReasons.stOuterTimeOutValidation.sMetsDisplayCode;
		aOuterStatus[1].stOACData.OuterRejectID := stOuterRejectReasons.stOuterTimeOutValidation.nRejectID;

		eState := E_OUTER_DONE_OCV;
END_IF

(* rising edge of bExecute *)
CASE eState OF

	(* idle *)
	E_OUTER_IDLE_OCV:

		(* scan for completed Outer when OAC files are required *)
		IF fbExecute.Q = TRUE THEN

			bDone := FALSE;
			bBusy := TRUE;

			bReffedOCVExec 			:=FALSE;
			bPackDataFoundInStruct 	:=FALSE;
			sOCVRejectCode 			:= '';

			nTrigID					:= 0;
			nNewOuterTrigID := nNewOuterTrigID +1;
			(*MEMMOVE(ADR(aLogTrigID[1]), ADR(aLogTrigID[0]), SIZEOF(aLogTrigID) - SIZEOF(aLogTrigID[0]));*)

			MEMSET(ADR(aOuterStatus[1]), 16#00, SIZEOF(aOuterStatus[1]));
			MEMSET(ADR(stLastOuterStatus), 16#00, SIZEOF(stLastOuterStatus));

			sLastReadOuterBarcode :=  '';
			sLastReadConfPackCode1 :=  '' ;

			MEMSET(ADR(stPacksDataFromOCV1), 16#00, SIZEOF(stPacksDataFromOCV1));
			MEMSET(ADR(stPacksDataFromOCV2), 16#00, SIZEOF(stPacksDataFromOCV2));

			eState := E_OUTER_READ_OCV;

		ELSIF bExecute = FALSE THEN

			(* reset outputs *)
			bDone := FALSE;
			bBusy := FALSE;
		END_IF

	E_OUTER_READ_OCV:

		IF	stProductInstruction.bEnablePacks  THEN

			IF  stBarcodeConfirmationCameraLastCodes.aCodeData[1].strDataString <> ''  THEN

				IF NOT bReffedOCVExec THEN
					FOR nOuterIndex := 1 TO cMAX_OUTER_STATUS_QUEUE  DO

						IF aOCVPackStatus[nOuterIndex].stOACData.AggregationCodes[1] <> '' AND
							aOCVPackStatus[nOuterIndex].stOACData.AggregationCodes[1]   = stBarcodeConfirmationCameraLastCodes.aCodeData[1].strDataString  THEN

							IF NOT  aOCVPackStatus[nOuterIndex].nStatus.22 THEN
								aOuterStatus[1]	 := aOCVPackStatus[nOuterIndex];
								aOuterStatus[1].sDataSourceTracker	:= 'OCV1_AGG';
							ELSE
								aOuterStatus[1].sDataSourceTracker	:= 'BIT22_AGG';
							END_IF
							bPackDataFoundInStruct :=TRUE;
							EXIT;
						END_IF

					END_FOR
				END_IF

				IF bPackDataFoundInStruct AND nOuterIndex > 1 THEN
					nInhibitOCVRestore 			:=FALSE;

					FOR nPackIndex := 1 TO  aOCVPackStatus[nOuterIndex-1].stOACData.NumberOfPacks  DO
							IF aOCVPackStatus[nOuterIndex-1].aOACPackStatus[nPackIndex] <> 5  THEN
									nInhibitOCVRestore :=TRUE;
							END_IF
					END_FOR
				END_IF

				IF NOT bPackDataFoundInStruct  THEN
					bReffedOCVExec :=TRUE;

					IF fbOCVRefeed.bOCVFileFound1 THEN
						 aOuterStatus[1] := stPacksDataFromOCV1;
					END_IF

					IF  fbOCVRefeed.bOCVFileFound1 THEN

						IF  NOT aOuterStatus[1].nStatus.22 THEN
							aOuterStatus[1].sDataSourceTracker	:= 'OCV_FILE';
						ELSE
							MEMSET(ADR(aOuterStatus[1]), 16#00, SIZEOF(aOuterStatus[1]));
							aOuterStatus[1].sDataSourceTracker	:= 'BIT22_FILE';
						END_IF
					END_IF
				END_IF

				nTrigID	:= aOuterStatus[1].nTriggerID;


				IF nTrigID > 0  THEN

					aOuterStatus[1].bOuterPresent := TRUE;
					aOuterStatus[1].stOACData.OuterTimeStamp := F_SYSTEM_SystemTimeAsISO8601(stCTDateTime.sSystemTime, stCTDateTime.sUTCTimeZoneOffset );
					aOuterStatus[1].nStatus.8 :=TRUE;

					aOuterStatus[1].stOACData.RetailSKU := stProductInstruction.sRetailSKU;
					aOuterStatus[1].stOACData.OuterMachine.ProductionSite :=  stProductInstruction.sProductionSite;
					aOuterStatus[1].stOACData.OuterMachine.ProductionLine := stProductInstruction.sProductionLine;
					aOuterStatus[1].stOACData.BatchNumber := stProductInstruction.sBatchNumber;
					aOuterStatus[1].stOACData.CodingAndTrackingMode := stProductInstruction.nOpMode;
					aOuterStatus[1].stOACData.AcceptanceLevel := stProductInstruction.nAcceptanceLevel;
					aOuterStatus[1].stOACData.NumberOfPacks	:= stProductInstruction.nPacksPerOuter;

					sOCVRejectCode 		:= 'OK';
					nOCVRejectID 			:= 0;

					eState := E_OUTER_BUILD_OAC_DATA;

				ELSIF  fbOCVRefeed.bTimeOut OR	(fbOCVRefeed.bDone AND NOT fbOCVRefeed.bOCVFileOK) THEN

					bReffedOCVExec :=FALSE;

					(*aOuterStatus[1].stOACData.AggregationCodes[1]   := stBarcodeConfirmationCameraLastCodes.aCodeData[1].strDataString;*)

					aOuterStatus[1].stOACData.OuterTimeStamp := F_SYSTEM_SystemTimeAsISO8601(stCTDateTime.sSystemTime, stCTDateTime.sUTCTimeZoneOffset );
					aOuterStatus[1].stOACData.RetailSKU := stProductInstruction.sRetailSKU;
					aOuterStatus[1].stOACData.OuterMachine.ProductionSite :=  stProductInstruction.sProductionSite;
					aOuterStatus[1].stOACData.OuterMachine.ProductionLine := stProductInstruction.sProductionLine;
					aOuterStatus[1].stOACData.BatchNumber := stProductInstruction.sBatchNumber;
					aOuterStatus[1].stOACData.CodingAndTrackingMode := stProductInstruction.nOpMode;

					aOuterStatus[1].stOACData.AcceptanceLevel := stProductInstruction.nAcceptanceLevel;
					aOuterStatus[1].stOACData.NumberOfPacks	:= stProductInstruction.nPacksPerOuter;

					sOCVRejectCode 	:=	stOuterRejectReasons.stOuterPackCodeDataNotFound.sMetsDisplayCode;
					nOCVRejectID		:=	stOuterRejectReasons.stOuterPackCodeDataNotFound.nRejectID;

					aOuterStatus[1].sDataSourceTracker	:= 'NO_FILE';
					nErrorCounter1 := nErrorCounter1+1;

					eState := E_OUTER_BUILD_OAC_DATA;
				END_IF
			ELSE

				aOuterStatus[1].stOACData.OuterTimeStamp :=F_SYSTEM_SystemTimeAsISO8601(stCTDateTime.sSystemTime, stCTDateTime.sUTCTimeZoneOffset );

				aOuterStatus[1].stOACData.RetailSKU := stProductInstruction.sRetailSKU;
				aOuterStatus[1].stOACData.OuterMachine.ProductionSite :=  stProductInstruction.sProductionSite;
				aOuterStatus[1].stOACData.OuterMachine.ProductionLine := stProductInstruction.sProductionLine;
				aOuterStatus[1].stOACData.BatchNumber := stProductInstruction.sBatchNumber;
				aOuterStatus[1].stOACData.CodingAndTrackingMode := stProductInstruction.nOpMode;

				(* load pack data for Outer *)
				aOuterStatus[1].stOACData.AcceptanceLevel := stProductInstruction.nAcceptanceLevel;
				aOuterStatus[1].stOACData.NumberOfPacks	:= stProductInstruction.nPacksPerOuter;
				aOuterStatus[1].sDataSourceTracker	:= 'ERR';

				nErrorCounter2 := nErrorCounter2+1;

				eState := E_OUTER_BUILD_OAC_DATA;
			END_IF
		ELSE

			aOuterStatus[1].stOACData.AggregationCodes[1]   := stBarcodeConfirmationCameraLastCodes.aCodeData[1].strDataString;

			aOuterStatus[1].stOACData.OuterTimeStamp := F_SYSTEM_SystemTimeAsISO8601(stCTDateTime.sSystemTime, stCTDateTime.sUTCTimeZoneOffset );
			aOuterStatus[1].stOACData.RetailSKU := stProductInstruction.sRetailSKU;
			aOuterStatus[1].stOACData.OuterMachine.ProductionSite :=  stProductInstruction.sProductionSite;
			aOuterStatus[1].stOACData.OuterMachine.ProductionLine := stProductInstruction.sProductionLine;
			aOuterStatus[1].stOACData.BatchNumber := stProductInstruction.sBatchNumber;
			aOuterStatus[1].stOACData.CodingAndTrackingMode := stProductInstruction.nOpMode;
			aOuterStatus[1].sDataSourceTracker	:= 'OUT_CS';

			sOCVRejectCode 		:= 'OK';
			nOCVRejectID			:= 0;

			eState := E_OUTER_BUILD_OAC_DATA;
		END_IF

	E_OUTER_BUILD_OAC_DATA:

		aOuterStatus[1].stOACData.ProductionDate := F_StringWildcard('#YYYYMMDD#', stSystemTime);
		aOuterStatus[1].stOACData.ProductionTime := F_StringWildcard('#hhmmss#', stSystemTime);
		aOuterStatus[1].stOACData.ProductionTimeOffset := F_SYSTEM_SystemTimeOffsetToHHMM(stCTDateTime.nSystemTimeOffset);


(********************************************************************************************************************************)
		(*IF stBarcodeConfirmationCameraLastCodes.sCodeData[1].strDataString <> ''  THEN

			aOuterStatus[1].bLabelApplied := TRUE;
			aOuterStatus[1].stOACData.Barcode := stBarcodeConfirmationCameraLastCodes.sCodeData[1].strDataString;

		ELSIF sOCVRejectCode ='OK'  THEN

			sOCVRejectCode	:=	stOuterRejectReasons.stOuterBarcodeNotRead.sMetsDisplayCode;
			nOCVRejectID		:=	stOuterRejectReasons.stOuterBarcodeNotRead.nRejectID;

		ELSIF nOCVRejectID = stOuterRejectReasons.stOuterConfirmCodeNotRead.nRejectID THEN

			sOCVRejectCode	:=	stOuterRejectReasons.stOuterGeneralCodeError.sMetsDisplayCode;
			nOCVRejectID		:=	stOuterRejectReasons.stOuterGeneralCodeError.nRejectID;
		END_IF*)

(********************************************************************************************************************************)
		(*IF aOuterStatus[1].stOACData.AggregationCodes[1] <> ''  THEN

			aOuterStatus[1].bLabelApplied := TRUE;
			aOuterStatus[1].stOACData.Barcode := aOuterStatus[1].stOACData.AggregationCodes[1];

		ELSIF stBarcodeConfirmationCameraLastCodes.aCodeData[1].strDataString = ''  THEN

			sOCVRejectCode 	:=	stOuterRejectReasons.stOuterBarcodeNotRead.sMetsDisplayCode;
			nOCVRejectID		:=	stOuterRejectReasons.stOuterBarcodeNotRead.nRejectID;

		END_IF*)
(********************************************************************************************************************************)

		IF stBarcodeConfirmationCameraLastCodes.aCodeData[1].strDataString <> ''  THEN

			aOuterStatus[1].bLabelApplied := TRUE;
			aOuterStatus[1].stOACData.Barcode := stBarcodeConfirmationCameraLastCodes.aCodeData[1].strDataString;

		ELSIF stBarcodeConfirmationCameraLastCodes.aCodeData[1].strDataString = ''  THEN

			sOCVRejectCode 	:=	stOuterRejectReasons.stOuterBarcodeNotRead.sMetsDisplayCode;
			nOCVRejectID		:=	stOuterRejectReasons.stOuterBarcodeNotRead.nRejectID;

		END_IF
(********************************************************************************************************************************)


		IF bQAReject THEN
			aOuterStatus[1].bQAReject 	:= 	bQAReject;
		END_IF

		aOuterStatus[1].nStatus.9 						:= TRUE;
		aOuterStatus[1].nTriggerID 					:= nNewOuterTrigID;
		aOuterStatus[1].stOACData.OuterRejectCode	:= sOCVRejectCode;
		aOuterStatus[1].stOACData.OuterRejectID		:= nOCVRejectID;

		eState := E_OUTER_DONE_OCV;

	E_OUTER_DONE_OCV:

		nOutersCompleted := nOutersCompleted + 1;
		stLastOuterStatus := aOuterStatus[1];

		MEMSET(ADR(stOuterStatusHMI), 16#00, SIZEOF(stOuterStatusHMI));

		stOuterStatusHMI.aAggregationCodes[1] := aOuterStatus[1].stOACData.AggregationCodes[1];

		stOuterStatusHMI.aAggregationCodesPosition[1] := 0;
		stOuterStatusHMI.aAggregationCodesPosition[2] := 0;

		sLastReadOuterBarcode :=  stBarcodeConfirmationCameraLastCodes.aCodeData[1].strDataString ;
		sLastReadConfPackCode1 :=  aOuterStatus[1].stOACData.AggregationCodes[1];

		MEMMOVE(ADR(aLogTimer[1]), ADR(aLogTimer), SIZEOF(aLogTimer)-SIZEOF(aLogTimer[1]));
		aLogTimer[0] :=tonTestTimer.ET;

		bReffedOCVExec :=FALSE;

		bDone := TRUE;
		bBusy := FALSE;

		eState := E_OUTER_IDLE_OCV;
ELSE

	eState := E_OUTER_IDLE_OCV;

END_CASE

aOCVFileCodeName[1]	:=	F_CodeToHex(F_CODE_GetItem(stBarcodeConfirmationCameraLastCodes.aCodeData[1].strDataString , eCodeAIType.SerialCode,
												SEL(bUseInterimCodeForValidation  , stMachineConfig.stCodeInfo_Pack, stMachineConfig.stCodeInfo_Intermediate)));
aOCVFileCodeName[2]	:=	F_CodeToHex(F_CODE_GetItem(stBarcodeConfirmationCameraLastCodes.aCodeData[2].strDataString , eCodeAIType.SerialCode,   stMachineConfig.stCodeInfo_Pack)); (*no reason to have 2 diffrent intermediate codes*)

fbOCVRefeed(
		bExecute 				:= bReffedOCVExec,
		aOCVFileCodeName 	:= aOCVFileCodeName,
		sTargetPath 			:= sLocalOCVPath,
		bSingleFileOnly		:= TRUE,
		tTimeout 				:= t#1s,
		stOuterStatus1 		=> stPacksDataFromOCV1,
		stOuterStatus2 		=> stPacksDataFromOCV2
		);

END_FUNCTION_BLOCK

// ---- POUs/_Exclude/FB_OUTER_RefeedOCVFilesWtihError.TcPOU
FUNCTION_BLOCK FB_OUTER_RefeedOCVFilesWtihError
VAR_INPUT
	bExecute				: BOOL;
	aOCVFileCodeName	: ARRAY[1..2] OF T_MaxString;
	sTargetPath			: STRING(50);		(* target OCV folder path *)
	tTimeout				: TIME;
	bSingleFileOnly		: BOOL;
END_VAR
VAR_OUTPUT

	bDone					: BOOL;
	bTimeOut				: BOOL;

	stOuterStatus1			: ST_OUTER_Status;
	stOuterStatus2			: ST_OUTER_Status;
	bOCVFileOK			: BOOL;
	bOCVFileFound1		: BOOL;
	bOCVFileFound2		: BOOL;
	sOCVFile1				: T_OCV_Filename;
	sOCVFile2				: T_OCV_Filename;

END_VAR
VAR
	fbOCVRefeed			: ARRAY[1..2] OF FB_OCV_FindFileWithError;
	fbExecute				: R_TRIG;
	tonTimoeOut			: TON;
END_VAR

fbExecute(CLK := bExecute);

IF fbExecute.Q = TRUE THEN

		MEMSET(ADR(stOuterStatus1), 16#00, SIZEOF(stOuterStatus1));
		MEMSET(ADR(stOuterStatus2), 16#00, SIZEOF(stOuterStatus2));


		sOCVFile1			:= '';			(* OCV filename *)
		sOCVFile2			:= '';			(* OCV filename *)


ELSIF NOT bExecute THEN

		MEMSET(ADR(stOuterStatus1), 16#00, SIZEOF(stOuterStatus1));
		MEMSET(ADR(stOuterStatus2), 16#00, SIZEOF(stOuterStatus2));

END_IF


fbOCVRefeed[1](
	bExecute			:= bExecute,
	strPackCode		:= aOCVFileCodeName[1],
	strLocalOCVPath	:= sTargetPath,
	sOuterStatus		:= stOuterStatus1,
	strOCVFile				=> sOCVFile1,
	nReadOCVError		=> nReadOCVError,
	nReadOCVFound		=> nReadOCVFound,
	nReadOCVFoundInErr	=> nReadOCVFoundInErr

);

bOCVFileFound1 := fbOCVRefeed[1].bOCVFileFound OR fbOCVRefeed[1].bOCVErrorFileFound;

fbOCVRefeed[2](
	bExecute			:= fbOCVRefeed[1].bDone AND NOT bOCVFileFound1 AND NOT bSingleFileOnly,
	strPackCode		:= aOCVFileCodeName[2],
	strLocalOCVPath	:= sTargetPath,
	sOuterStatus		:= stOuterStatus2,
	strOCVFile				=> sOCVFile2,
	nReadOCVError		=> nReadOCVError,
	nReadOCVFound		=> nReadOCVFound,
	nReadOCVFoundInErr	=> nReadOCVFoundInErr

);

bOCVFileFound2 := fbOCVRefeed[2].bOCVFileFound OR fbOCVRefeed[2].bOCVErrorFileFound;

(*****************outputs**********************)
IF bSingleFileOnly THEN
	bDone			:= fbOCVRefeed[1].bDone;
	bOCVFileOK 	:= bOCVFileFound1;
ELSE
	bDone			:= fbOCVRefeed[2].bDone;
	bOCVFileOK 	:= bOCVFileFound2;
END_IF

tonTimoeOut(
	IN				:= bExecute AND NOT bOCVFileFound1 AND NOT bOCVFileFound2,
	PT				:= tTimeOut,
	Q				=> bTimeOut
);

END_FUNCTION_BLOCK

// ---- POUs/_Exclude/OCV FBs/FB_OCV_FindFileWithError.TcPOU
(* converts strOuterBarcode to OCV filename and loads data *)
FUNCTION_BLOCK FB_OCV_FindFileWithError
VAR_INPUT
	bExecute			: BOOL;		(* set TRUE to load OCV file *)
	strPackCode	 	: STRING(255);	(* Outer barcode *)
	strLocalOCVPath	: STRING(50);(* local OCv path *)
END_VAR
VAR_IN_OUT
	sOuterStatus			: ST_OUTER_Status;	(* Outer status *)
END_VAR
VAR_OUTPUT
	bDone				: BOOL;		(* TRUE = find file complete *)
	bBusy				: BOOL;		(* TRUE = find file in progress *)
	bError				: BOOL;		(* TRUE = error occurred *)
	nErrorID				: UDINT;	(* error code *)
	bOCVFileFound 		: BOOL;
	bOCVErrorFileFound		: BOOL;		(* TRUE = OCv file found *)
	strOCVFile			: T_OCV_Filename;	(* OCV filename *)
	strOCVErrorFile		: T_OCV_Filename;	(* OCV filename *)
	strOCVErrorNameFound	: T_OCV_Filename;	(* OCV filename *)
	nReadOCVError		: UDINT;
	nReadOCVFound		: UDINT;
	nReadOCVFoundInErr	: UDINT;
END_VAR
VAR
	fbExecute				: R_TRIG;
	eState				: E_OCV_State;
	eErrorState			: E_OCV_State;

	fbReadFile			: FB_XmlSrvRead;
	fbGetNewFileInfo		: FB_FILE_GetFileInfo;
	fbReadErrorFile		: FB_XmlSrvRead;

END_VAR

fbExecute(CLK := bExecute);

CASE eState OF

	(* idle *)
	E_OCV_IDLE:

	(* rising edge of bExecute *)
	IF fbExecute.Q = TRUE THEN

		(* initialise outputs *)
		bDone := FALSE;
		bBusy := TRUE;
		bError := FALSE;
		nErrorID := 0;
		strOCVFile := '';
		strOCVErrorFile :='';

		(* convert strOuterBarcode to OCV filename *)
		bOCVFileFound 		:= FALSE;
		bOCVErrorFileFound		:= FALSE;

		MEMSET(ADR(sOuterStatus), 16#00, SIZEOF(sOuterStatus));

		strOCVFile := 	 F_CONCAT3('OCV_',strPackCode, '.xml');
		strOCVErrorFile := 	 F_CONCAT3('*',strPackCode, '*');

		strOCVErrorNameFound	:= '';

		eState := E_OCV_READFILE;

	(* bExecute has been reset *)
	ELSIF bExecute = FALSE THEN

		(* reset outputs *)
		bDone := FALSE;
		bBusy := FALSE;
		bError := FALSE;
		nErrorID := 0;

		bOCVFileFound 		:= FALSE;
		bOCVErrorFileFound		:= FALSE;

		strOCVErrorNameFound	:= '';

	END_IF

(* read good OCV  file *)
	E_OCV_READFILE:

		fbReadFile(
			sNetId		:= '',
			ePath		:= PATH_GENERIC,
			nMode		:= XMLSRV_SKIPMISSING,
			pSymAddr	:= ADR(sOuterStatus),
			cbSymSize	:= SIZEOF(sOuterStatus),
			sFilePath	:= CONCAT(strLocalOCVPath, strOCVFile),
			sXPath		:= '/OCVPack',
			bExecute	:= TRUE,
			tTimeout	:= T#1s
		);
		
		(* read file complete *)
		IF fbReadFile.bBusy = FALSE THEN
		
			(* read file completed OK *)
			IF fbReadFile.bError = FALSE THEN

				nReadOCVFound := nReadOCVFound + 1;
				(* OAC file exists *)
				bOCVFileFound := TRUE;

				eState := E_OCV_DONE;
			(* read file failed *)
			ELSE
		
				(* update outputs *)
				bError := TRUE;
				nErrorID := fbReadFile.nErrId;
				eErrorState := eState;
				nReadOCVError :=nReadOCVError + 1;
				eState := E_OCV_FINDFILE;
		
			END_IF

			(* close off fbReadFile *)
			fbReadFile(bExecute := FALSE);
		END_IF

	E_OCV_FINDFILE:


		fbGetNewFileInfo(
			bExecute			:=TRUE,			(* set TRUE to get file info *)
			strPathSource		:=CONCAT(strLocalOCVPath,'Error\'),	(* folder path for SOURCE file, wildcard chars '*' and '?' can be used *)
			strFileName		:=strOCVErrorFile,	(* name of file to be copied, wildcard chars '*' and '?' can be used *)
			tTimeout			:=t#1s
					);	(* full name of file found *)

		(* delete file complete *)
		IF fbGetNewFileInfo.bBusy = FALSE THEN

			(* delete file completed OK *)
			IF fbGetNewFileInfo.bError = FALSE THEN

				IF fbGetNewFileInfo.bFileExists THEN
					strOCVErrorNameFound := fbGetNewFileInfo.strFileFound;
					bOCVErrorFileFound := TRUE;
					eState := E_OCV_READERRORFILE;
				ELSE
					eState := E_OCV_DONE;
				END_IF
			(* copy file error *)
			ELSE
				(* no error has previously occurred *)
				IF bError = FALSE THEN

					(* log error code and failure state *)
					bError := TRUE;
					nErrorID := fbGetNewFileInfo.nErrorID;
					eErrorState := eState;
				END_IF

				eState := E_OCV_DONE;

			END_IF

			(* close off fbDeleteFile *)
			fbGetNewFileInfo(bExecute := FALSE);
		END_IF
	(* read error OCV  file *)
	E_OCV_READERRORFILE:

		fbReadErrorFile(
			sNetId		:= '',
			ePath		:= PATH_GENERIC,
			nMode		:= XMLSRV_SKIPMISSING,
			pSymAddr	:= ADR(sOuterStatus),
			cbSymSize	:= SIZEOF(sOuterStatus),
			sFilePath	:= F_CONCAT3(strLocalOCVPath, 'Error\', strOCVErrorNameFound),
			sXPath		:= '/OCVPack',
			bExecute	:= TRUE,
			tTimeout	:= T#1s
		);
		
		(* read file complete *)
		IF fbReadErrorFile.bBusy = FALSE THEN
		
			(* read file completed OK *)
			IF fbReadErrorFile.bError = FALSE THEN

				nReadOCVFoundInErr := nReadOCVFoundInErr + 1;
				(* OAC file exists *)
				bOCVErrorFileFound := TRUE;
		
				eState := E_OCV_DONE;
			(* read file failed *)
			ELSE
		
				(* update outputs *)
				bError := TRUE;
				nErrorID := fbReadErrorFile.nErrId;
				eErrorState := eState;
				nReadOCVError :=nReadOCVError + 1;
				eState := E_OCV_DONE;

			END_IF

			(* close off fbReadFile *)
			fbReadErrorFile(bExecute := FALSE);
		END_IF

	(* complete *)
	E_OCV_DONE:

		(* update outputs *)
		bDone := TRUE;
		bBusy := FALSE;

		eState := E_OCV_IDLE;


(* unknown state *)
ELSE

	eState := E_OCV_IDLE;

	(* clear outputs *)
	bDone := FALSE;
	bBusy := FALSE;
	bError := FALSE;
	nErrorID := 0;
	bOCVFileFound 		:= FALSE;
	bOCVErrorFileFound		:= FALSE;

	strOCVErrorNameFound	:= '';
END_CASE

END_FUNCTION_BLOCK

// ---- POUs/_Exclude/FB_OUTER_CompleteDataFromOCV.TcPOU
 FUNCTION_BLOCK FB_OUTER_CompleteDataFromOCV
VAR_INPUT
	bExecute								: BOOL;		(* set TRUE to scan arrOuterStatus for completed Outers *)
	bValidationTimeout					: BOOL;
	bOuterCameraDone					: BOOL;
	bConfirmationCameraDone			: BOOL;
	stOuterValidationCameraLastCodes	: ST_SCANNER_ImageData;
	stPackConfirmationCameraLastCodes	: ST_SCANNER_ImageData;
	nPackPos1								: INT 	:=1;
	nPackPos2								: INT	:=2;
	bUseInterimCodeForValidation		: BOOL;
	sLocalOCVPath							: STRING(255);
	stCTDateTime							: ST_SYSTEM_DateTime;	(* CaseTrace date/time structure *)
	bQAReject								: BOOL;
END_VAR
VAR_IN_OUT
	stProductInstruction		: ST_PCM_Status;					(* Product Instruction *)
	stOuterRejectReasons		: ST_RejectReasonsForOuter;
	aOuterStatus				: ARRAY[1..cMAX_OUTER_STATUS_QUEUE] OF ST_OUTER_Status;	(* Outer status register *)
	aOCVPackStatus			: ARRAY[1..cMAX_OUTER_STATUS_QUEUE] OF ST_OUTER_Status;	(* Outer status register *)
	stOuterStatusHMI			: ST_HMI_OuterStatus;
END_VAR
VAR_OUTPUT
	bDone						: BOOL;			(* TRUE = validation complete *)
	bBusy						: BOOL;			(* TRUE = validation in progress *)

	stLastOuterStatus			: ST_OUTER_Status;

	sLastReadOuterBarcode	: T_OUTER_Barcode;
	sLastReadConfPackCode1	: T_PACK_Barcode;
	sLastReadConfPackCode2 	: T_PACK_Barcode;
	(*aConfPackCodeInPosition		: ARRAY[0..1] OF T_PACK_Barcode;*)
	sOCVRejectCode			: T_RejectCode;
	nOCVRejectID				: UINT;
	bPackDataFoundInStruct	: BOOL;
	nInhibitOCVRestore		: BOOL;
	bReadyToOCVResotre		: BOOL;
	nOutersCompleted			: UDINT;

END_VAR
VAR
	eState						: E_OUTER_AgrregationState;
	fbExecute					: R_TRIG;
	fbTimeOut					: R_TRIG;
	stSystemTime				: TIMESTRUCT;

	(*nAggregartionPackCode	: INT;*)

	nOuterIndex				: INT;
	(*nMaxOuterIndex				: INT;*)
	nPackIndex				: INT;

	aOCVFileCodeName		: ARRAY[1..2] OF T_MaxString;
	bReffedOCVExec			: BOOL;
	fbOCVRefeed				: FB_OUTER_RefeedOCVFilesWtihError; (*FB_PACK_RefeedOCVFilesWtihError;*)

	stPacksDataFromOCV1	: ST_OUTER_Status;
	stPacksDataFromOCV2	: ST_OUTER_Status;

	nTrigID						: UDINT;
	aLogTrigID					: ARRAY[0..5] OF UDINT;
	nNewOuterTrigID			: UDINT;

	(*aPackStatusValue				: ARRAY[0..10] OF INT;
	aRejectCodePointer            		: ARRAY[0..10] OF STRING(10);

	fbValidatePack					: FB_CODE_ValidateExplicitCode;*)

	nErrorCounter1			: INT;
	nErrorCounter2			: INT;
	nErrorCounter3			: INT;

	tonTestTimer				: TON;
	aLogTimer 					: ARRAY[0..100] OF TIME;
END_VAR

fbExecute(CLK := bExecute);
fbTimeOut(CLK := bValidationTimeout);

stSystemTime := stCTDateTime.sSystemTime;

tonTestTimer(In:= bBusy AND NOT bDone, PT:= t#5000ms);
IF fbTimeOut.Q THEN

		aOuterStatus[1].stOACData.ProductionDate := F_StringWildcard('#YYYYMMDD#', stSystemTime);
		aOuterStatus[1].stOACData.ProductionTime := F_StringWildcard('#hhmmss#', stSystemTime);
		aOuterStatus[1].stOACData.ProductionTimeOffset := F_SYSTEM_SystemTimeOffsetToHHMM(stCTDateTime.nSystemTimeOffset);

		aOuterStatus[1].stOACData.OuterTimeStamp :=F_SYSTEM_SystemTimeAsISO8601(stCTDateTime.sSystemTime, stCTDateTime.sUTCTimeZoneOffset );
		aOuterStatus[1].stOACData.RetailSKU := stProductInstruction.sRetailSKU;
		aOuterStatus[1].stOACData.OuterMachine.ProductionSite :=  stProductInstruction.sProductionSite;
		aOuterStatus[1].stOACData.OuterMachine.ProductionLine := stProductInstruction.sProductionLine;
		aOuterStatus[1].stOACData.BatchNumber := stProductInstruction.sBatchNumber;
		aOuterStatus[1].stOACData.CodingAndTrackingMode := stProductInstruction.nOpMode;

		aOuterStatus[1].stOACData.AcceptanceLevel := stProductInstruction.nAcceptanceLevel;
		aOuterStatus[1].stOACData.NumberOfPacks	:= stProductInstruction.nPacksPerOuter;

		IF NOT bOuterCameraDone AND NOT bConfirmationCameraDone THEN
			aOuterStatus[1].sDataSourceTracker	:= 'T_OUT_ALL';
		ELSIF NOT bOuterCameraDone THEN
			aOuterStatus[1].sDataSourceTracker	:= 'T_OUT_OVC';
		ELSIF NOT bConfirmationCameraDone	THEN
			aOuterStatus[1].sDataSourceTracker	:= 'T_OUT_PCC';
		ELSE
			aOuterStatus[1].sDataSourceTracker	:= 'T_OUT_FB';
		END_IF

		aOuterStatus[1].nStatus.9 := TRUE;
		aOuterStatus[1].nTriggerID := nNewOuterTrigID;
		aOuterStatus[1].stOACData.OuterRejectCode := stOuterRejectReasons.stOuterTimeOutValidation.sMetsDisplayCode;
		aOuterStatus[1].stOACData.OuterRejectID := stOuterRejectReasons.stOuterTimeOutValidation.nRejectID;

		eState := E_OUTER_DONE_OCV;
END_IF

(* rising edge of bExecute *)
CASE eState OF

	(* idle *)
	E_OUTER_IDLE_OCV:

		(* scan for completed Outer when OAC files are required *)
		IF fbExecute.Q = TRUE THEN

			bDone := FALSE;
			bBusy := TRUE;

			bReffedOCVExec 			:=FALSE;
			bPackDataFoundInStruct 	:=FALSE;
			sOCVRejectCode 			:= '';

			nTrigID					:= 0;
			nNewOuterTrigID := nNewOuterTrigID +1;
			MEMMOVE(ADR(aLogTrigID[1]), ADR(aLogTrigID[0]), SIZEOF(aLogTrigID) - SIZEOF(aLogTrigID[0]));

			MEMSET(ADR(aOuterStatus[1]), 16#00, SIZEOF(aOuterStatus[1]));
			MEMSET(ADR(stLastOuterStatus), 16#00, SIZEOF(stLastOuterStatus));

			MEMSET(ADR(stPacksDataFromOCV1), 16#00, SIZEOF(stPacksDataFromOCV1));
			MEMSET(ADR(stPacksDataFromOCV2), 16#00, SIZEOF(stPacksDataFromOCV2));

			eState := E_OUTER_READ_OCV;

		ELSIF bExecute = FALSE THEN

			(* reset outputs *)
			bDone := FALSE;
			bBusy := FALSE;
		END_IF

	E_OUTER_READ_OCV:

		IF	stProductInstruction.bEnablePacks  THEN

			IF  stPackConfirmationCameraLastCodes.aCodeData[1].strDataString <> '' OR  stPackConfirmationCameraLastCodes.aCodeData[2].strDataString <> '' THEN

				IF NOT bReffedOCVExec THEN
					FOR nOuterIndex := 1 TO cMAX_OUTER_STATUS_QUEUE  DO

						IF aOCVPackStatus[nOuterIndex].stOACData.AggregationCodes[1] <> '' AND
							(aOCVPackStatus[nOuterIndex].stOACData.AggregationCodes[1]   = stPackConfirmationCameraLastCodes.aCodeData[1].strDataString 	OR
				 			aOCVPackStatus[nOuterIndex].stOACData.AggregationCodes[1]  = stPackConfirmationCameraLastCodes.aCodeData[2].strDataString) THEN

							IF NOT  aOCVPackStatus[nOuterIndex].nStatus.22 THEN
								aOuterStatus[1]	 := aOCVPackStatus[nOuterIndex];
								aOuterStatus[1].sDataSourceTracker	:= 'OCV1_AGG';
							ELSE
								aOuterStatus[1].sDataSourceTracker	:= 'BIT22_AGG';
							END_IF
							bPackDataFoundInStruct :=TRUE;
							EXIT;

						ELSIF aOCVPackStatus[nOuterIndex].stOACData.AggregationCodes[2] <> '' AND nPackPos2 <> 0 AND
							(aOCVPackStatus[nOuterIndex].stOACData.AggregationCodes[2]   = stPackConfirmationCameraLastCodes.aCodeData[1].strDataString 	OR
				 			aOCVPackStatus[nOuterIndex].stOACData.AggregationCodes[2]  = stPackConfirmationCameraLastCodes .aCodeData[2].strDataString) THEN

							IF NOT  aOCVPackStatus[nOuterIndex].nStatus.22 THEN
								aOuterStatus[1]	 := aOCVPackStatus[nOuterIndex];
								aOuterStatus[1].sDataSourceTracker	:= 'OCV2_AGG';
							ELSE
								aOuterStatus[1].sDataSourceTracker	:= 'BIT22_AGG';
							END_IF
							bPackDataFoundInStruct :=TRUE;
							EXIT;
						END_IF

					END_FOR
				END_IF

				IF bPackDataFoundInStruct AND nOuterIndex > 1 THEN
					nInhibitOCVRestore 			:=FALSE;

					FOR nPackIndex := 1 TO  aOCVPackStatus[nOuterIndex-1].stOACData.NumberOfPacks  DO
							IF aOCVPackStatus[nOuterIndex-1].aOACPackStatus[nPackIndex] <> 5  THEN
									nInhibitOCVRestore :=TRUE;
							END_IF
					END_FOR
				END_IF

				IF NOT bPackDataFoundInStruct  THEN
					bReffedOCVExec :=TRUE;

					IF fbOCVRefeed.bOCVFileFound1 THEN
						 aOuterStatus[1] := stPacksDataFromOCV1;

					ELSIF fbOCVRefeed.bOCVFileFound2 AND nPackPos2 <> 0 THEN
						 aOuterStatus[1] := stPacksDataFromOCV2;
					END_IF

					IF  fbOCVRefeed.bOCVFileFound1 OR  fbOCVRefeed.bOCVFileFound2 THEN

						IF  NOT aOuterStatus[1].nStatus.22 THEN
							aOuterStatus[1].sDataSourceTracker	:= 'OCV_FILE';
						ELSE
							MEMSET(ADR(aOuterStatus[1]), 16#00, SIZEOF(aOuterStatus[1]));
							aOuterStatus[1].sDataSourceTracker	:= 'BIT22_FILE';
						END_IF
					END_IF
				END_IF

				nTrigID	:= aOuterStatus[1].nTriggerID;

				aLogTrigID[0] := nTrigID;

				IF (aLogTrigID[1] -  aLogTrigID[2] = 1) AND (aLogTrigID[2] -  aLogTrigID[3] = 1) AND (aLogTrigID[3] -  aLogTrigID[4] = 1) AND (aLogTrigID[4] -  aLogTrigID[5] = 1) THEN
					bReadyToOCVResotre	:= TRUE;
				ELSE
					bReadyToOCVResotre	:= FALSE;
				END_IF

				IF nTrigID > 0  THEN

					aOuterStatus[1].bOuterPresent := TRUE;
					aOuterStatus[1].stOACData.OuterTimeStamp := F_SYSTEM_SystemTimeAsISO8601(stCTDateTime.sSystemTime, stCTDateTime.sUTCTimeZoneOffset );
					aOuterStatus[1].nStatus.8 :=TRUE;

					aOuterStatus[1].stOACData.RetailSKU := stProductInstruction.sRetailSKU;
					aOuterStatus[1].stOACData.OuterMachine.ProductionSite :=  stProductInstruction.sProductionSite;
					aOuterStatus[1].stOACData.OuterMachine.ProductionLine := stProductInstruction.sProductionLine;
					aOuterStatus[1].stOACData.BatchNumber := stProductInstruction.sBatchNumber;
					aOuterStatus[1].stOACData.CodingAndTrackingMode := stProductInstruction.nOpMode;
					aOuterStatus[1].stOACData.AcceptanceLevel := stProductInstruction.nAcceptanceLevel;
					aOuterStatus[1].stOACData.NumberOfPacks	:= stProductInstruction.nPacksPerOuter;

					sOCVRejectCode 		:= 'OK';
					nOCVRejectID 			:= 0;

					eState := E_OUTER_BUILD_OAC_DATA;

				ELSIF  fbOCVRefeed.bTimeOut OR	(fbOCVRefeed.bDone AND NOT fbOCVRefeed.bOCVFileOK) THEN

					bReffedOCVExec :=FALSE;

					aOuterStatus[1].stOACData.OuterTimeStamp := F_SYSTEM_SystemTimeAsISO8601(stCTDateTime.sSystemTime, stCTDateTime.sUTCTimeZoneOffset );
					aOuterStatus[1].stOACData.RetailSKU := stProductInstruction.sRetailSKU;
					aOuterStatus[1].stOACData.OuterMachine.ProductionSite :=  stProductInstruction.sProductionSite;
					aOuterStatus[1].stOACData.OuterMachine.ProductionLine := stProductInstruction.sProductionLine;
					aOuterStatus[1].stOACData.BatchNumber := stProductInstruction.sBatchNumber;
					aOuterStatus[1].stOACData.CodingAndTrackingMode := stProductInstruction.nOpMode;

					aOuterStatus[1].stOACData.AcceptanceLevel := stProductInstruction.nAcceptanceLevel;
					aOuterStatus[1].stOACData.NumberOfPacks	:= stProductInstruction.nPacksPerOuter;

					sOCVRejectCode 	:=	stOuterRejectReasons.stOuterPackCodeDataNotFound.sMetsDisplayCode;
					nOCVRejectID		:=	stOuterRejectReasons.stOuterPackCodeDataNotFound.nRejectID;

					aOuterStatus[1].sDataSourceTracker	:= 'NO_FILE';
					nErrorCounter1 := nErrorCounter1+1;

					eState := E_OUTER_BUILD_OAC_DATA;
				END_IF
			ELSE

				aOuterStatus[1].stOACData.OuterTimeStamp :=F_SYSTEM_SystemTimeAsISO8601(stCTDateTime.sSystemTime, stCTDateTime.sUTCTimeZoneOffset );

				IF NOT nInhibitOCVRestore AND bReadyToOCVResotre THEN
					aOuterStatus[1].nStatus.16 :=TRUE;
				END_IF

				aOuterStatus[1].stOACData.RetailSKU := stProductInstruction.sRetailSKU;
				aOuterStatus[1].stOACData.OuterMachine.ProductionSite :=  stProductInstruction.sProductionSite;
				aOuterStatus[1].stOACData.OuterMachine.ProductionLine := stProductInstruction.sProductionLine;
				aOuterStatus[1].stOACData.BatchNumber := stProductInstruction.sBatchNumber;
				aOuterStatus[1].stOACData.CodingAndTrackingMode := stProductInstruction.nOpMode;

				(* load pack data for Outer *)
				aOuterStatus[1].stOACData.AcceptanceLevel := stProductInstruction.nAcceptanceLevel;
				aOuterStatus[1].stOACData.NumberOfPacks	:= stProductInstruction.nPacksPerOuter;
				aOuterStatus[1].sDataSourceTracker	:= 'ERR';

				nErrorCounter2 := nErrorCounter2+1;

				sOCVRejectCode 	:=	stOuterRejectReasons.stOuterConfirmCodeNotRead.sMetsDisplayCode;
				nOCVRejectID		:=	stOuterRejectReasons.stOuterConfirmCodeNotRead.nRejectID;

				eState := E_OUTER_BUILD_OAC_DATA;
			END_IF
		ELSE

			aOuterStatus[1].stOACData.OuterTimeStamp := F_SYSTEM_SystemTimeAsISO8601(stCTDateTime.sSystemTime, stCTDateTime.sUTCTimeZoneOffset );
			aOuterStatus[1].stOACData.RetailSKU := stProductInstruction.sRetailSKU;
			aOuterStatus[1].stOACData.OuterMachine.ProductionSite :=  stProductInstruction.sProductionSite;
			aOuterStatus[1].stOACData.OuterMachine.ProductionLine := stProductInstruction.sProductionLine;
			aOuterStatus[1].stOACData.BatchNumber := stProductInstruction.sBatchNumber;
			aOuterStatus[1].stOACData.CodingAndTrackingMode := stProductInstruction.nOpMode;
			aOuterStatus[1].sDataSourceTracker	:= 'OUT_CS';

			sOCVRejectCode 		:= 'OK';
			nOCVRejectID			:= 0;

			eState := E_OUTER_BUILD_OAC_DATA;
		END_IF

	E_OUTER_BUILD_OAC_DATA:

		aOuterStatus[1].stOACData.ProductionDate := F_StringWildcard('#YYYYMMDD#', stSystemTime);
		aOuterStatus[1].stOACData.ProductionTime := F_StringWildcard('#hhmmss#', stSystemTime);
		aOuterStatus[1].stOACData.ProductionTimeOffset := F_SYSTEM_SystemTimeOffsetToHHMM(stCTDateTime.nSystemTimeOffset);

		IF stOuterValidationCameraLastCodes.aCodeData[1].strDataString  <>''  THEN

			aOuterStatus[1].bLabelApplied := TRUE;
			aOuterStatus[1].stOACData.Barcode := stOuterValidationCameraLastCodes.aCodeData[1].strDataString;

			IF stOuterValidationCameraLastCodes.aCodeData[1].nProgramNo = 2 THEN
				nRecoverOuterLable	:= nRecoverOuterLable +1;
			END_IF

		ELSIF sOCVRejectCode ='OK'  THEN

			sOCVRejectCode	:=	stOuterRejectReasons.stOuterBarcodeNotRead.sMetsDisplayCode;
			nOCVRejectID		:=	stOuterRejectReasons.stOuterBarcodeNotRead.nRejectID;

		ELSIF nOCVRejectID = stOuterRejectReasons.stOuterConfirmCodeNotRead.nRejectID THEN

			sOCVRejectCode	:=	stOuterRejectReasons.stOuterGeneralCodeError.sMetsDisplayCode;
			nOCVRejectID		:=	stOuterRejectReasons.stOuterGeneralCodeError.nRejectID;
		END_IF

		IF stOuterValidationCameraLastCodes.aCodeData[1].strDataString  = ''  THEN
			nErrorCounter3	 := nErrorCounter3	+1;
		END_IF

		IF bQAReject THEN
			aOuterStatus[1].bQAReject 	:= 	bQAReject;
		END_IF

		aOuterStatus[1].nStatus.9 						:= TRUE;
		aOuterStatus[1].nTriggerID 					:= nNewOuterTrigID;
		aOuterStatus[1].stOACData.OuterRejectCode	:= sOCVRejectCode;
		aOuterStatus[1].stOACData.OuterRejectID		:= nOCVRejectID;

		eState := E_OUTER_DONE_OCV;

	E_OUTER_DONE_OCV:

		nOutersCompleted := nOutersCompleted + 1;
		stLastOuterStatus := aOuterStatus[1];

		MEMSET(ADR(stOuterStatusHMI), 16#00, SIZEOF(stOuterStatusHMI));

		IF stPackConfirmationCameraLastCodes.aCodeData[1].nProgramNo = 1 THEN
			stOuterStatusHMI.aAggregationCodes[SEL(stMachineConfig.bFirstPackCodeOnTop, 2,1)] := stPackConfirmationCameraLastCodes.aCodeData[1].strDataString;
			stOuterStatusHMI.aAggregationCodes[SEL(stMachineConfig.bFirstPackCodeOnTop, 1,2)] := stPackConfirmationCameraLastCodes.aCodeData[2].strDataString;
		ELSIF stPackConfirmationCameraLastCodes.aCodeData[1].nProgramNo = 2 THEN
			stOuterStatusHMI.aAggregationCodes[SEL(stMachineConfig.bFirstPackCodeOnTop, 1,2)] := stPackConfirmationCameraLastCodes.aCodeData[1].strDataString;
			stOuterStatusHMI.aAggregationCodes[SEL(stMachineConfig.bFirstPackCodeOnTop, 2,1)] := stPackConfirmationCameraLastCodes.aCodeData[2].strDataString;
		END_IF
		stOuterStatusHMI.aAggregationCodesPosition[1] := nPackPos1;
		stOuterStatusHMI.aAggregationCodesPosition[2] := nPackPos2;

		sLastReadOuterBarcode	:=  stOuterValidationCameraLastCodes.aCodeData[1].strDataString;
		sLastReadConfPackCode1 :=  stPackConfirmationCameraLastCodes.aCodeData[1].strDataString ;
		sLastReadConfPackCode2 	:=  stPackConfirmationCameraLastCodes.aCodeData[2].strDataString ;

		MEMMOVE(ADR(aLogTimer[1]), ADR(aLogTimer), SIZEOF(aLogTimer)-SIZEOF(aLogTimer[1]));
		aLogTimer[0] :=tonTestTimer.ET;

		bReffedOCVExec :=FALSE;

		bDone := TRUE;
		bBusy := FALSE;

		eState := E_OUTER_IDLE_OCV;
ELSE

	eState := E_OUTER_IDLE_OCV;

END_CASE

aOCVFileCodeName[1]	:=	F_CodeToHex(F_CODE_GetItem(stPackConfirmationCameraLastCodes.aCodeData[1].strDataString , eCodeAIType.SerialCode,
												SEL(bUseInterimCodeForValidation  , stMachineConfig.stCodeInfo_Pack, stMachineConfig.stCodeInfo_Intermediate)));
aOCVFileCodeName[2]	:=	F_CodeToHex(F_CODE_GetItem(stPackConfirmationCameraLastCodes.aCodeData[2].strDataString , eCodeAIType.SerialCode,   stMachineConfig.stCodeInfo_Pack)); (*no reason to have 2 diffrent intermediate codes*)

fbOCVRefeed(
		bExecute 				:= bReffedOCVExec,
		aOCVFileCodeName 	:= aOCVFileCodeName,
		sTargetPath 			:= sLocalOCVPath,
		bSingleFileOnly		:= (nPackPos2	= 0),
		tTimeout 				:= t#1s,
		stOuterStatus1 		=> stPacksDataFromOCV1,
		stOuterStatus2 		=> stPacksDataFromOCV2
		);

END_FUNCTION_BLOCK

// ---- POUs/_Exclude/FB_OUTER_RepairOCVContent.TcPOU
FUNCTION_BLOCK FB_OUTER_RepairOCVContent
VAR_INPUT
	bExecute					: BOOL;			(* scan for completed Outer *)
	ePackAggregationMode	: E_SYSTEM_PackAggregationMode ;
	bResetErrorStats			: BOOL;
	strLocalOCVPath			: STRING(255);		(* OCV folder path *)
	sProductInstruction			: ST_PCM_Status;
	nPackPos1				: INT 	:=1;
	nPackPos2				: INT	:=2;
	bUseInterimCodeForValidation	: BOOL;
	stDuplicatedItem			: ST_RejectItems;(*stPackRejectReasons.stPackCodesDuplicated*)
	bEnableSUPICheck			: BOOL;
	nSUPI_Identyfication		: DINT;
	tTimeout					: TIME := t#1s;
END_VAR
VAR_IN_OUT
	strNewPackCodeRefeed		:T_PACK_Barcode;
	arrErrorOuters				: ARRAY[1..cMAX_OUTER_STATUS_QUEUE] OF ST_OUTER_Status;
	nErrorIndex				: INT;
	arrOCVPackStatus			: ARRAY[1..cMAX_OUTER_STATUS_QUEUE] OF ST_OUTER_Status;
	stOCVDataDB					: ST_DB_OCVDataCtrl;
	stCodeInfo_Pack			: ST_CodeInfo;
	stCodeInfo_Intermediate		: ST_CodeInfo;
END_VAR
VAR_OUTPUT
	bDone					: BOOL;			(* TRUE = validation complete *)
	bBusy					: BOOL;			(* TRUE = validation in progress *)
	bError					: BOOL;			(* TRUE = validation error *)
	nErrorID					: UDINT;			(* error ID *)
	strOCVFile1				: T_OCV_Filename;	(* OCV file name *)
	strOCVFile2				: T_OCV_Filename;	(* OCV file name *)
	nOutersStoredInOCV		: UINT;
END_VAR
VAR
	fbExecute					: R_TRIG;
	tonTimeOut				: TON;
	eState					: E_OUTER_State;
	fbDuplicatesPackCodesDB		: FB_PACK_DuplicatesPackCodesDB;
	aOCVFileCodeName			: ARRAY[1..2] OF T_MaxString;
	fbWriteOCVFile			: FB_OCV_WriteFile;
	fbValidatePack				: FB_CODE_ValidateExplicitCode;

	sErrorOuterData			: ST_OUTER_Status;	(* Outer status array *)
	sEmptyOuterData			: ST_OUTER_Status;	(* Outer status array *)


	bAggregationCodes1Valid			: BOOL;
	bAggregationCodes2Valid			: BOOL;

	nPackIndex				: INT;
	nSourceIndex				: INT;

	nOuterIndex				: INT;
	nMaxOuterIndex 			: INT;
	bPackDataRemovedFromST	: BOOL;

	nStatusError				: UDINT;
	nValidationError			: UDINT;
	nEmptySource				: UDINT;

	nWriteOCVerror			: UDINT;
	strMemoPackCodeRefeed	:T_PACK_Barcode;

	(*Diagnostic counters*)
	aDiagCounter : ARRAY[0..5] OF INT;

END_VAR

(* monitor rising edge of bExecute *)
fbExecute(CLK := bExecute);

(* monitor Busy timeout *)
tonTimeOut(IN:=bBusy, PT:=tTimeout, Q=>);

IF tonTimeOut.Q THEN
	bError := TRUE;
	nErrorID := 10;
	strNewPackCodeRefeed := '';
	eState := E_OUTER_IDLE;
END_IF

IF bResetErrorStats THEN

	(* clear error statistic counters *)
	nStatusError := 0;
	nValidationError := 0;
	nEmptySource := 0;
	nOutersStoredInOCV := 0;
	nWriteOCVerror := 0;
	strMemoPackCodeRefeed := '';
END_IF

(* rising edge of bExecute *)
CASE eState OF

	(* idle *)
	E_OUTER_IDLE:

		(* scan for completed Outer when OAC files are required *)
		IF fbExecute.Q = TRUE THEN

			(* update outputs *)
			bDone := FALSE;
			bBusy := TRUE;
			bError := FALSE;
			nErrorID := 0;

			aDiagCounter[0] := aDiagCounter[0] +1;

			eState := E_OUTER_SCAN;

		(* no action required *)
		ELSIF bExecute = FALSE THEN

			(* reset outputs *)
			bDone := FALSE;
			bBusy := FALSE;
			bError := FALSE;
			(*bAggregationCodes1Valid := FALSE;
			bAggregationCodes2Valid := FALSE;
			fbWriteOCVFile(bExecute := FALSE);
			nErrorID := 0;*)

		END_IF

	(* scan for completed Outer *)
	E_OUTER_SCAN:

		bBusy := TRUE;
		nSourceIndex := 0;
		sErrorOuterData := arrErrorOuters[nErrorIndex];

		IF sProductInstruction.nPacksPerOuter - sErrorOuterData.stOACData.NumberOfLinkedPacks = 1  AND strNewPackCodeRefeed <> '' THEN

			FOR nPackIndex := 1 TO sProductInstruction.nPacksPerOuter BY 1 DO

				IF  sErrorOuterData.aOACPackStatus[nPackIndex] = 0 OR sErrorOuterData.aOACPackStatus[nPackIndex] = 1  THEN

						nSourceIndex := nPackIndex;
					EXIT;

				END_IF

			END_FOR

		END_IF


		IF nSourceIndex > 0 THEN

			aDiagCounter[1] := aDiagCounter[1] +1;

			MEMSET(ADR(aOCVFileCodeName), 16#00, SIZEOF(aOCVFileCodeName));

			fbValidatePack(	sFullCode := strNewPackCodeRefeed,
							stCodeInfo := stMachineConfig.stCodeInfo_Pack,
							stProductInstruction := sProductInstruction);


			IF fbValidatePack.bValidationOK THEN

				sErrorOuterData.stOACData.PackCode[nSourceIndex]:= strNewPackCodeRefeed;
				sErrorOuterData.stOACData.PackCodeStatus[nSourceIndex].6 := TRUE;

				aDiagCounter[2] := aDiagCounter[2] +1;

				(*fbChekcDupPackCode(nNumberPackInOuters := sProductInstruction.nPacksPerOuter,
							sOuterStatus := sErrorOuterData,
							stDuplicatedItem := stDuplicatedItem,
							bDuplicateFound => 	);*)

				fbDuplicatesPackCodesDB(
					stDuplicatedItem := stDuplicatedItem,
					bExtendedDupCheck	:=	FALSE,
					stOuterStatus := sErrorOuterData,
					stLastOuterStatus := sEmptyOuterData,
					bDuplicateFound =>
					);

				(*IF bEnableSUPICheck AND  nSUPI_Identyfication <> 0  THEN
					sErrorOuterData.aPackSUPIResult[nSourceIndex]	:=  F_CogCheck(sErrorOuterData.stOACData.PackCode[nSourceIndex]);
					IF  sErrorOuterData.aPackSUPIResult[nSourceIndex] <>  nSUPI_Identyfication   THEN
						sErrorOuterData.nStatus.26 := TRUE;
						sErrorOuterData.aOACPackStatus[nSourceIndex]:= 2;
					END_IF
				END_IF*)

				IF NOT sErrorOuterData.nStatus.23 (*AND NOT sErrorOuterData.nStatus.26*) THEN


					sErrorOuterData.aOACPackStatus[nSourceIndex]:= 5;
					sErrorOuterData.stOACData.PackRejectCode[nSourceIndex]:= 'OK';
					sErrorOuterData.stOACData.PackRejectID[nSourceIndex]	:= 0;

					IF nPackPos1= nSourceIndex AND sErrorOuterData.stOACData.AggregationCodes[1] = '' THEN sErrorOuterData.stOACData.AggregationCodes[1] := strNewPackCodeRefeed; END_IF
					IF nPackPos2= nSourceIndex AND sErrorOuterData.stOACData.AggregationCodes[2] = '' THEN sErrorOuterData.stOACData.AggregationCodes[2] := strNewPackCodeRefeed; END_IF

					sErrorOuterData.aPackCodes[nSourceIndex].sBuffer[1].strCode := sErrorOuterData.stOACData.PackCode[nSourceIndex];
					sErrorOuterData.aPackCodes[nSourceIndex].sBuffer[1].nStatus := sErrorOuterData.aOACPackStatus[nSourceIndex];
					sErrorOuterData.aPackCodes[nSourceIndex].sBuffer[1].nStringSize := LEN(sErrorOuterData.stOACData.PackCode[nSourceIndex]);
					sErrorOuterData.aPackCodes[nSourceIndex].sBuffer[2].strCode := sErrorOuterData.stOACData.PackCode[nSourceIndex];
					sErrorOuterData.aPackCodes[nSourceIndex].sBuffer[2].nStatus := sErrorOuterData.aOACPackStatus[nSourceIndex];
					sErrorOuterData.aPackCodes[nSourceIndex].sBuffer[2].nStringSize := LEN(sErrorOuterData.stOACData.PackCode[nSourceIndex]);

					sErrorOuterData.stOACData.NumberOfLinkedPacks := sProductInstruction.nPacksPerOuter;

					aDiagCounter[3] := aDiagCounter[3] +1;

					eState := E_OUTER_CHECKPACKS;
				ELSE
					sErrorOuterData.stOACData.PackCode[nSourceIndex]:= 'STATUS REJECTED';

					nStatusError := nStatusError+1;
					strNewPackCodeRefeed := '';
					bError := TRUE;
					nErrorID := 1;

					eState := E_OUTER_IDLE;
				END_IF
			ELSE
				sErrorOuterData.stOACData.PackCode[nSourceIndex]:= 'CODE INVALIDE';
				sErrorOuterData.aOACPackStatus[nSourceIndex]:= 2;

				nValidationError := nValidationError+1;
				strNewPackCodeRefeed := '';

				bError := TRUE;
				nErrorID := 2;


				eState := E_OUTER_IDLE;
			END_IF

		ELSE
			nEmptySource := nEmptySource+1;
			strNewPackCodeRefeed := '';

			bError := TRUE;
			nErrorID := 3;

			eState := E_OUTER_IDLE;
		END_IF

	E_OUTER_CHECKPACKS:

		nMaxOuterIndex := UDINT_TO_INT(SIZEOF(arrOCVPackStatus) / SIZEOF(arrOCVPackStatus[1]));
		bPackDataRemovedFromST := FALSE;

		FOR nPackIndex := 1 TO sProductInstruction.nPacksPerOuter BY 1 DO
			IF nPackIndex  <> nSourceIndex  THEN
				FOR nOuterIndex := 1 TO nMaxOuterIndex BY 1 DO

					IF arrOCVPackStatus[nOuterIndex].stOACData.PackCode[nPackIndex] = sErrorOuterData.stOACData.PackCode[nPackIndex] THEN

						MEMMOVE(ADR(arrOCVPackStatus[nOuterIndex]), ADR(arrOCVPackStatus[nOuterIndex + 1]), SIZEOF(arrOCVPackStatus[1]) * (nMaxOuterIndex - nOuterIndex) );
						MEMSET(ADR(arrOCVPackStatus[nMaxOuterIndex]), 0, SIZEOF(arrOCVPackStatus[1]));
						bPackDataRemovedFromST := TRUE;
						EXIT;
					END_IF

				END_FOR
			END_IF
			IF bPackDataRemovedFromST THEN
				EXIT;
			END_IF
		END_FOR

		eState := E_OUTER_WRITEDATA;












	(* write OCVC file *)
	E_OUTER_WRITEDATA:

		aDiagCounter[4] := aDiagCounter[4] +1;

		aOCVFileCodeName[1]	:=	F_CodeToHex(F_CODE_GetItem(sErrorOuterData.stOACData.AggregationCodes[1] , eCodeAIType.SerialCode,
																				SEL(bUseInterimCodeForValidation, stCodeInfo_Pack, stCodeInfo_Intermediate)));
		aOCVFileCodeName[2]	:=	F_CodeToHex(F_CODE_GetItem(sErrorOuterData.stOACData.AggregationCodes[2] , eCodeAIType.SerialCode,   stCodeInfo_Pack)); (*no reason to have 2 diffrent intermediate codes*)

		IF F_InvalidateASCIIChar(aOCVFileCodeName[1]) =	0 	THEN bAggregationCodes1Valid := nPackPos1 <> 0 OR  bUseInterimCodeForValidation;  	END_IF
		IF F_InvalidateASCIIChar(aOCVFileCodeName[2]) =	0 	THEN bAggregationCodes2Valid := nPackPos2 <> 0; 		END_IF

		(* write OCV file *)
		fbWriteOCVFile(
			bExecute					:= TRUE,
			sTargetPath				:= strLocalOCVPath,
			ePackAggregationMode	:= ePackAggregationMode,
			nPacksPerOuter			:= sProductInstruction.nPacksPerOuter,
			aOCVFileCodeName		:= aOCVFileCodeName,  (*strAggregationCodes is a table*)
			bSkipWriteFile1			:= NOT bAggregationCodes1Valid,
			bSkipWriteFile2			:= NOT bAggregationCodes2Valid,
			stOCVPackStatus			:= sErrorOuterData
			);

		(* write OCV file complete *)
		IF fbWriteOCVFile.bDone = TRUE THEN

			(* write OCV file completed OK *)
			IF fbWriteOCVFile.bError = FALSE THEN

				arrErrorOuters[nErrorIndex].aOACPackStatus[nSourceIndex]:= 6;

				arrErrorOuters[nErrorIndex].stOACData.PackCode[nSourceIndex]:= strNewPackCodeRefeed;
				arrErrorOuters[nErrorIndex].stOACData.PackRejectCode[nSourceIndex]:= 'OCV Restored';
				arrErrorOuters[nErrorIndex].stOACData.PackRejectID[nSourceIndex]:= 0;

				arrErrorOuters[nErrorIndex].stOACData.NumberOfLinkedPacks := sProductInstruction.nPacksPerOuter;
				arrErrorOuters[nErrorIndex].stOACData.OuterRejectCode := CONCAT(arrErrorOuters[nErrorIndex].stOACData.OuterRejectCode, ' *OCV Restored*');
				arrErrorOuters[nErrorIndex].stOACData.OuterRejectID := 0;

				(* count OCV files written *)
				nOutersStoredInOCV := nOutersStoredInOCV + 1;
				aDiagCounter[5] := aDiagCounter[5] +1;

				strOCVFile1 := fbWriteOCVFile.sOCVFile1;
				strOCVFile2 := fbWriteOCVFile.sOCVFile2;
				eState := E_OUTER_DONE;

			ELSE
				(* update sOuterStatus - OCV file write error  - general error for OCV *)
				nWriteOCVerror := nWriteOCVerror +1;
				strNewPackCodeRefeed := '';

				bError := TRUE;
				nErrorID := 4;

				eState := E_OUTER_IDLE;
			END_IF

			(* close off fbWriteOCVFile*)
			fbWriteOCVFile(bExecute := FALSE);
		END_IF

	(* OCV file complete *)
	E_OUTER_DONE:

		strMemoPackCodeRefeed := strNewPackCodeRefeed;
		strNewPackCodeRefeed := '';

		(* update outputs *)
		bDone := TRUE;
		bBusy := FALSE;

		eState := E_OUTER_IDLE;

(* unknown state *)
ELSE
	eState := E_OUTER_IDLE;
END_CASE

END_FUNCTION_BLOCK

// ---- POUs/_Exclude/FB_OUTER_WriteOACFileLoop.TcPOU
(* scan and validate Outers, generate OAC file for new valid Outers *)
FUNCTION_BLOCK FB_OUTER_WriteOACFileLoop
VAR_INPUT
	bExecute					: BOOL;			(* scan for completed Outer *)
	strLocalOACPath			: STRING(50);	(* TEMP folder path *)
	nPacksPerOuter			: INT;
	nCodingAndTrackingMode	: INT;
	stCTDateTime				: ST_SYSTEM_DateTime;
	bDisableCompareOAC		: BOOL;
	(*sMetsSearchCode	: STRING(50);   stPackRejectReasons.stPackCodesSUPIError.sMetsSearchCode*)
END_VAR
VAR_IN_OUT
	stCodeInfo_Pack	: ST_CodeInfo;
	stCodeInfo_Outer	: ST_CodeInfo;
	aOuterStatus		: ARRAY[1..cMAX_OUTER_STATUS_QUEUE] OF ST_OUTER_Status;	(* Outer status array *)
	stLastOuterStatus	: ST_OUTER_Status;
END_VAR
VAR_OUTPUT
	bDone				: BOOL;			(* TRUE = validation complete *)
	bBusy				: BOOL;			(* TRUE = validation in progress *)
	bError				: BOOL;			(* TRUE = validation error *)
	nErrorID				: UDINT;		(* error ID *)
	nOACFiles			: UDINT;		(* OAC files created *)
	strOACFile			: T_OAC_Filename;	(* OAC file name *)
	sDeletedOACFile		: T_OAC_Filename;	(* OAC file name *)
	sOuterStatus			: ST_OUTER_Status;	(* Outer status *)
	bWriteOACError		: UINT;
	bInvalidOAC			: BOOL;
	bOACDupBacroceFound	: BOOL;
	bOACDupPacksFound	: BOOL;
	nOACFilesDeleted 		: UINT;
	bOACUpdated			: BOOL;
	sCodesAggregatedToOAC	: T_LongSTRING;
END_VAR
VAR
	fbExecute				: R_TRIG;
	eState				: E_OUTER_State;
	nMaxOuterIndex		: INT;
	nOuterIndex			: INT;
	nSourceIndex			: INT;
	fbWriteOACFile		: FB_OAC_WriteFile;

	eCodeAIType			: E_CodeAIType;

	sBarcode				: T_OUTER_Barcode;
	bInvalidBarcode		: BOOL;
	nInvalidErrorCounter	: UINT;
	sInvalidLastCode		: T_OUTER_Barcode;

	nPackCodeDupIndex	: UINT;
	nPackCodeCheckIndex	: UINT;

	strOACFileToMove		: T_OAC_Filename;	(* OAC file name *)
	fbMoveOACFile		: FB_FILE_MoveWithDate;

	arrLocalOuterStatus			: ARRAY[1..10] OF  ST_OUTER_Status;
	nCounter :UDINT;

	nOACLogIndex			: UINT;

END_VAR

(* monitor rising edge of bExecute *)
fbExecute(CLK := bExecute);

(* rising edge of bExecute *)
CASE eState OF

	(* idle *)
	E_OUTER_IDLE:

		(* scan for completed Outer when OAC files are required *)
		IF fbExecute.Q = TRUE THEN

			(* update outputs *)
			bDone := FALSE;
			bBusy := TRUE;
			bError := FALSE;
			nErrorID := 0;

			(* clear outputs *)
			nOACFiles := 0;

			(* max Outer index *)
			nMaxOuterIndex := UDINT_TO_INT(SIZEOF(aOuterStatus) / SIZEOF(aOuterStatus[1]));

			eState := E_OUTER_SCAN;

		(* no action required *)
		ELSIF bExecute = FALSE THEN

			(* reset outputs *)
			bDone := FALSE;
			bBusy := FALSE;
			bError := FALSE;
			nErrorID := 0;
		END_IF


	(* scan for completed Outer *)
	E_OUTER_SCAN:

		(* reset index of Outer to be written to OAC file *)
		nSourceIndex 			:= 0;

		sBarcode					:= '';
		bInvalidBarcode			:= FALSE;
		bInvalidOAC				:= FALSE;
		bOACDupBacroceFound	:= FALSE;
		bOACDupPacksFound		:= FALSE;

		bOACUpdated				:= FALSE;
		sCodesAggregatedToOAC	:= '';

		(* scan aOuterStatus  backward - ensures that oldest Outer will be written first *)
		FOR nOuterIndex := nMaxOuterIndex TO 1 BY -1 DO

			(* TriggerID > 0 indicates Outer data present -  *)
			IF aOuterStatus[nOuterIndex].nTriggerID > 0 AND
				aOuterStatus[nOuterIndex].stOACData.CodingAndTrackingMode >= 7 AND
				(aOuterStatus[nOuterIndex].nStatus.10  OR
					(aOuterStatus[nOuterIndex].nStatus.11 AND aOuterStatus[nOuterIndex].nStatus.14)) AND
				NOT aOuterStatus[nOuterIndex].nStatus.12 AND
				NOT aOuterStatus[nOuterIndex].nStatus.13 THEN

				(* log index of Outer requiring OAC file *)
				nSourceIndex := nOuterIndex;
				EXIT;
			END_IF
		END_FOR

		(* Outer found requiring OAC file to be written *)
		IF nSourceIndex > 0 THEN

			(* copy Outer data from aOuterStatus *)
			sOuterStatus := aOuterStatus[nSourceIndex];

			A_CheckOACData();

			IF bInvalidBarcode THEN

				bError := TRUE;
				nErrorID := 666;
				nInvalidErrorCounter:=nInvalidErrorCounter+1;
				sInvalidLastCode	:= sBarcode;

				sOuterStatus.nStatus.13 := TRUE;

				eState := E_OUTER_STATUS;

			ELSIF bInvalidOAC AND (bOACDupBacroceFound OR bOACDupPacksFound) THEN

				eState := E_OUTER_DELETEFILE;
			ELSE
				eState := E_OUTER_WRITEDATA;
			END_IF
		(* no OAC files required *)
		ELSE

			eState := E_OUTER_DONE;
		END_IF

	(* delete OAC to error folder *)
	E_OUTER_DELETEFILE:

		strOACFileToMove := F_CONCAT3('OAC_', F_OUTER_BarcodeToHex(aOuterStatus[nSourceIndex +1].stOACData.Barcode), '.xml');

		(* delete OAC file *)
		fbMoveOACFile(
				bExecute			:= TRUE,
				strPathSource		:= strLocalOACPath,
				strPathTarget		:= CONCAT(strLocalOACPath,'Error\' ),
				strFileName		:= strOACFileToMove,
				stCTDateTime		:= stCTDateTime,
				tTimeout			:= cHALF_SECOND
		);

		(* delete file complete *)
		IF NOT fbMoveOACFile.bBusy  THEN

			(* delete  file completed OK *)
			IF NOT  fbMoveOACFile.bError THEN

				(* update counter *)
				nOACFilesDeleted := nOACFilesDeleted + 1;
				sDeletedOACFile := fbMoveOACFile.strLastFileMoved;

			(* delete command error or file not found *)
			ELSE

				bError := TRUE;
				nErrorID := fbMoveOACFile.nErrorID + 1000;

			END_IF

			(* close off fbDeleteOACFile *)
			fbMoveOACFile(bExecute := FALSE);

			eState := E_OUTER_WRITEDATA;
		END_IF

	(* write OAC file *)
	E_OUTER_WRITEDATA:

		(* write OAC file *)
		fbWriteOACFile(
			bExecute					:= TRUE,
			sLocalOACPath				:= strLocalOACPath,
			bInvalidOAC				:= bInvalidOAC,
			bOACDupBacroceFound	:= bOACDupBacroceFound,
			bOACDupPacksFound		:= bOACDupPacksFound,
			stCTDateTime				:= stCTDateTime,
			stOACData					:= sOuterStatus.stOACData,
			tTimeout					:= cHALF_SECOND,
		);

		(* write OAC file complete *)
		IF fbWriteOACFile.bDone = TRUE THEN

			strOACFile := fbWriteOACFile.sOACFile;

			(* write OAC file completed OK *)
			IF fbWriteOACFile.bError = FALSE THEN

				(* count OAC files written *)
				nOACFiles := nOACFiles + 1;

				(* update sOuterStatus - OAC file written OK *)
				sOuterStatus.nStatus.12 := TRUE;

			(* write OAC file error *)
			ELSE
				bError := TRUE;
				nErrorID := fbWriteOACFile.nErrorID + 2000;

				bWriteOACError:=bWriteOACError+1;
				(* update sOuterStatus - OAC file write error *)
				sOuterStatus.stOACData.OuterCodeStatus.6 := TRUE;
				sOuterStatus.nStatus.13 := TRUE;
			END_IF

			eState := E_OUTER_STATUS;

			(* close off fbWriteOACFile*)
			fbWriteOACFile(bExecute := FALSE);
		END_IF


	(* update Outer status *)
	E_OUTER_STATUS:

		(* move sOuterStatus data back to shift reg *)
		FOR nOuterIndex := nMaxOuterIndex TO 1 BY -1 DO

			(* matching nTriggerID found *)
			IF aOuterStatus[nOuterIndex].nTriggerID = sOuterStatus.nTriggerID AND
				NOT aOuterStatus[nOuterIndex].nStatus.12 AND NOT aOuterStatus[nOuterIndex].nStatus.13 THEN


				nCounter := nCounter +1;
		(*!*)	stLastOuterStatus :=sOuterStatus;
				MEMMOVE(ADR(arrLocalOuterStatus[2]), ADR(arrLocalOuterStatus[1]), SIZEOF(arrLocalOuterStatus)-SIZEOF(arrLocalOuterStatus[1]));
				arrLocalOuterStatus[1] :=stLastOuterStatus;

				(* move updated Outer data to shift reg *)
				aOuterStatus[nOuterIndex] := sOuterStatus;

				sCodesAggregatedToOAC := F_CONCAT3(aOuterStatus[nOuterIndex].stOACData.OuterRejectCode,' - ',  F_CODE_GetItem(aOuterStatus[nOuterIndex].stOACData.Barcode, eCodeAIType.SerialCode, stCodeInfo_Outer));
				sCodesAggregatedToOAC := F_CONCAT6(sCodesAggregatedToOAC,'	[', RIGHT(aOuterStatus[nOuterIndex] .stOACData.AggregationCodes[1],7),']:[',RIGHT(aOuterStatus[nOuterIndex] .stOACData.AggregationCodes[2],7),']');

				FOR nOACLogIndex := 1 TO MIN(nPacksPerOuter ,cMAX_PACKS_PER_OUTER) BY 1 DO
					sCodesAggregatedToOAC :=F_LongCONCAT(sCodesAggregatedToOAC, '     ');
					sCodesAggregatedToOAC := F_LongCONCAT(sCodesAggregatedToOAC, RIGHT(F_CODE_GetItem(aOuterStatus[nOuterIndex] .stOACData.PackCode[nOACLogIndex], eCodeAIType.SerialCode, stCodeInfo_Pack),7));
				END_FOR

				bOACUpdated := TRUE;
				EXIT;
			END_IF
		END_FOR

		eState := E_OUTER_SCAN;

	(* OAC file complete *)
	E_OUTER_DONE:

		(* update outputs *)
		bDone := TRUE;
		bBusy := FALSE;

		eState := E_OUTER_IDLE;


(* unknown state *)
ELSE

	eState := E_OUTER_IDLE;
END_CASE

ACTION A_CheckOACData:
sBarcode:= F_CODE_GetItem(sOuterStatus.stOACData.Barcode, eCodeAIType.SerialCode, stCodeInfo_Outer);
bInvalidOAC := aOuterStatus[nOuterIndex].nStatus.11;

IF F_InvalidateASCIIChar(sBarcode) >  0 	THEN

	bInvalidBarcode := TRUE;

ELSIF	LEN(sBarcode) <> stCodeInfo_Outer.stSerialCode.nCodeLength AND stCodeInfo_Outer.stSerialCode.bValidate THEN

	bInvalidOAC := TRUE;
END_IF

IF NOT  bInvalidOAC  AND NOT bDisableCompareOAC  AND NOT bInvalidBarcode THEN


	IF sOuterStatus.stOACData.Barcode =  aOuterStatus[nSourceIndex +1].stOACData.Barcode AND
		LEN(aOuterStatus[nSourceIndex +1].stOACData.Barcode) >= stCodeInfo_Outer.nMinLength  THEN


		aOuterStatus[nSourceIndex +1].nStatus.22 := TRUE;
		aOuterStatus[nSourceIndex +1].stOACData.DataSource := 'REM';

		sOuterStatus.nStatus.22 := TRUE;
		sOuterStatus.stOACData.DataSource := 'REM';

		bInvalidOAC	 := TRUE;
		bOACDupBacroceFound := TRUE;
	END_IF

	IF NOT bOACDupBacroceFound THEN
		FOR nPackCodeCheckIndex:= 1 TO nPacksPerOuter DO
			FOR nPackCodeDupIndex := 1 TO nPacksPerOuter DO
				IF sOuterStatus.stOACData.PackCode[nPackCodeCheckIndex] <> '' AND aOuterStatus[nSourceIndex +1].nStatus.10  AND
					sOuterStatus.stOACData.PackCode[nPackCodeCheckIndex] =  aOuterStatus[nSourceIndex +1].stOACData.PackCode[nPackCodeDupIndex] THEN


					aOuterStatus[nSourceIndex +1].nStatus.22 := TRUE;
					aOuterStatus[nSourceIndex +1].stOACData.DataSource := 'REM';

					sOuterStatus.nStatus.22 := TRUE;
					sOuterStatus.stOACData.DataSource := 'REM';

					bInvalidOAC := TRUE;
					bOACDupPacksFound := TRUE;
					EXIT;
				END_IF
			END_FOR
			IF bOACDupPacksFound THEN
				EXIT;
			END_IF
		END_FOR
	END_IF
END_IF
END_ACTION

END_FUNCTION_BLOCK

// ---- POUs/_Exclude/FB_PACK_DuplicatesPackCodes.TcPOU
FUNCTION_BLOCK FB_PACK_DuplicatesPackCodes
VAR_INPUT
	nNumberPackInOuters					: INT;
	stDuplicatedItem						: ST_RejectItems;
END_VAR
VAR_OUTPUT
	bDuplicateFound 			: BOOL;
	sDuplicatePackCode			: T_PACK_Barcode;
END_VAR
VAR_IN_OUT
	sOuterStatus				: ST_OUTER_Status;	(* Outer status *)
END_VAR
VAR
	nCheckIndex : INT;
	nPackIndex : INT;
	nDuplicatePairs	: INT;
	(*nDupAmount		: INT;*)
	nGoodPackReads	: INT;
	nLastDuplicate		: INT;
END_VAR

nDuplicatePairs	:=0;
nGoodPackReads	:=nNumberPackInOuters;
bDuplicateFound 	:= FALSE;
sDuplicatePackCode := '';

	(* for all other Packs in Outer *)
FOR  nPackIndex :=1 TO cMAX_PACKS_PER_OUTER DO

	IF sOuterStatus.stOACData.PackCode[nPackIndex] <> ''
		AND sOuterStatus.stOACData.PackCode[nPackIndex] <> 'NOK'
		AND sOuterStatus.aOACPackStatus[nPackIndex] > 4 THEN

		FOR nCheckIndex := nPackIndex  TO cMAX_PACKS_PER_OUTER DO

			(* check Pack is not current Pack *)
			IF nCheckIndex <> nPackIndex  AND sOuterStatus.aOACPackStatus[nCheckIndex] <> 3
				AND sOuterStatus.stOACData.PackCode[nCheckIndex] <> ''
				AND  sOuterStatus.stOACData.PackCode[nCheckIndex] <> 'NOK' THEN
				(* currentpack code contains data and matches another pack code *)
				IF sOuterStatus.stOACData.PackCode[nPackIndex] = sOuterStatus.stOACData.PackCode[nCheckIndex]
					AND sOuterStatus.aOACPackStatus[nCheckIndex] > 4 THEN

					(* duplicate packs found *)
					sOuterStatus.aOACPackStatus[nPackIndex] := 3;
					sOuterStatus.aOACPackStatus[nCheckIndex] := 3;
					bDuplicateFound := TRUE;

					(*Counting how many different pairs found*)
					IF  sOuterStatus.stOACData.PackCode[nCheckIndex] <> sDuplicatePackCode THEN
						sDuplicatePackCode :=  sOuterStatus.stOACData.PackCode[nPackIndex];
						nDuplicatePairs := nDuplicatePairs + 1;
					END_IF

					sOuterStatus.stOACData.PackRejectCode[nPackIndex]  := stDuplicatedItem.sMetsDisplayCode;
	   				sOuterStatus.stOACData.PackRejectID[nPackIndex]  := stDuplicatedItem.nRejectID;
					sOuterStatus.stOACData.PackRejectCode[nCheckIndex]  := stDuplicatedItem.sMetsDisplayCode;
					sOuterStatus.stOACData.PackRejectID[nCheckIndex]  := stDuplicatedItem.nRejectID;

				END_IF
			END_IF

		END_FOR
	END_IF
END_FOR

IF bDuplicateFound THEN

	sOuterStatus.nStatus.23 := TRUE;
	nLastDuplicate := nLastDuplicate+1;

	FOR  nPackIndex :=1 TO cMAX_PACKS_PER_OUTER DO
		IF sOuterStatus.aOACPackStatus[nPackIndex] = 3 THEN nGoodPackReads := nGoodPackReads - 1; END_IF
	END_FOR

END_IF

END_FUNCTION_BLOCK

// ---- POUs/_Exclude/FB_PACK_ValidateOCVContent.TcPOU
FUNCTION_BLOCK FB_PACK_ValidateOCVContent
VAR_INPUT
	nOCVControlCheckStatus		: BYTE;
	nPacksPerOuter			: UINT;
	stCTDateTime				: ST_SYSTEM_DateTime;
	bUseIntermediateCode		: BOOL;
END_VAR
VAR_IN_OUT
	stCodeInfo_Pack			: ST_CodeInfo;
	stCodeInfo_Intermediate	: ST_CodeInfo;
	(*aInterimCodeQueue		: ARRAY[1..cMAX_INTERMEDIATE_CODE_QUEUE] OF T_MaxString;*)
	stOCVStatus				: ST_OUTER_Status;	(* Outer status *)
	stNextOCVStatus			: ST_OUTER_Status;	(* Next Outer status used for check duplicat in OCV queue *)
END_VAR
VAR_OUTPUT
	aOCVFileCodeName			: ARRAY[1..2] OF T_MaxString;
	aOCVFileCodeToDelete		: ARRAY[1..2] OF T_MaxString;
	bInvalidPackFound				: BOOL;
	bDuplicatePackFound			: BOOL;
	bDuplicateInterimFound			: BOOL;
	bMasterListFound				: BOOL;
	bEmptyAggregationCode		: BOOL;
END_VAR
VAR
	eCodeAIType				: E_CodeAIType;
	nPackCodeCheckIndex		: UINT;
	nPackCodeDupIndex		: UINT;
	nInterimCodeDupIndex	: UINT;
END_VAR

MEMSET(ADR(aOCVFileCodeName), 16#00, SIZEOF(aOCVFileCodeName));

bInvalidPackFound			:= FALSE;
bDuplicatePackFound 		:= FALSE;
bDuplicateInterimFound 	:= FALSE;
bMasterListFound			:= FALSE;
bEmptyAggregationCode 	:= FALSE;

IF nOCVControlCheckStatus = 0 THEN

	aOCVFileCodeName[1]	:=	F_CodeToHex(F_CODE_GetItem(stOCVStatus.stOACData.AggregationCodes[1] , eCodeAIType.SerialCode, SEL(bUseIntermediateCode, stCodeInfo_Pack, stCodeInfo_Intermediate)));
	aOCVFileCodeName[2]	:=	F_CodeToHex(F_CODE_GetItem(stOCVStatus.stOACData.AggregationCodes[2] , eCodeAIType.SerialCode,   stCodeInfo_Pack)); (*no reason to have 2 diffrent intermediate codes*)

ELSE
	MEMSET(ADR(aOCVFileCodeToDelete), 16#00, SIZEOF(aOCVFileCodeToDelete));

	IF stOCVStatus.stOACData.AggregationCodes[1] <>  cCODE_OVERWIRTTEN 	THEN
		aOCVFileCodeName[1]	:=	F_CODE_GetItem(stOCVStatus.stOACData.AggregationCodes[1] , eCodeAIType.SerialCode, SEL(bUseIntermediateCode, stCodeInfo_Pack, stCodeInfo_Intermediate));
	ELSE
		aOCVFileCodeName[1]	:= '';
	END_IF

	IF stOCVStatus.stOACData.AggregationCodes[2] <>  cCODE_OVERWIRTTEN 	THEN
		aOCVFileCodeName[2]	:=	F_CODE_GetItem(stOCVStatus.stOACData.AggregationCodes[2] , eCodeAIType.SerialCode,   stCodeInfo_Pack); (*no reason to have 2 diffrent intermediate codes*)
	ELSE
		aOCVFileCodeName[2]	:= '';
	END_IF

	IF nOCVControlCheckStatus.0 THEN

		(*DuplicatPackFound();*)
		DuplicateInterimFound();
	END_IF

	IF nOCVControlCheckStatus.1
		AND NOT bDuplicatePackFound
		AND NOT bDuplicateInterimFound	THEN

		InvalidPackFound();
	END_IF

	IF nOCVControlCheckStatus.2
		AND NOT bDuplicatePackFound
		AND NOT bDuplicateInterimFound
		AND NOT bInvalidPackFound	THEN

		MasterListFound();
	END_IF

	IF nOCVControlCheckStatus.3 THEN
		;
	END_IF

	IF nOCVControlCheckStatus.4 THEN
		;
	END_IF

	IF NOT bDuplicatePackFound AND NOT bDuplicateInterimFound AND NOT bMasterListFound  THEN

		aOCVFileCodeName[1] :=  F_CodeToHex(aOCVFileCodeName[1]);
		aOCVFileCodeName[2] :=  F_CodeToHex(aOCVFileCodeName[2]);
	END_IF

	IF aOCVFileCodeName[1] = '' AND aOCVFileCodeName[2] = '' THEN
		aOCVFileCodeName[1] := F_CONCAT3('EMPTY' ,'_' , F_SYSTEM_SystemTimeToCHM_Header(stCTDateTime.sSystemTime));

		bEmptyAggregationCode := TRUE;
	END_IF
END_IF

ACTION DuplicateInterimFound:
(*IF  stNextOCVStatus.nStatus.6
		AND bUseIntermediateCode
		AND stOCVStatus.stOACData.AggregationCodes[1] = stNextOCVStatus.stOACData.AggregationCodes[1]
		AND stOCVStatus.stOACData.AggregationCodes[1] <> cCODE_OVERWIRTTEN
		AND stOCVStatus.stOACData.AggregationCodes[1] <> ''					THEN

			aOCVFileCodeName[1] := CONCAT('DUP_INT_', F_CodeToHex(aOCVFileCodeName[1]));
			stOCVStatus.nStatus.22 := TRUE;
			stOCVStatus.sDataSourceTracker  := 'DUPLICAT';

			FOR nInterimCodeDupIndex := 1 TO cMAX_INTERMEDIATE_CODE_QUEUE DO
				aInterimCodeQueue[nInterimCodeDupIndex] 	:=	cCODE_OVERWIRTTEN;
			END_FOR

			bDuplicateInterimFound := TRUE;

END_IF
*)
IF stOCVStatus.sDataSourceTracker  = 'DUPLICAT' THEN

		aOCVFileCodeName[1] := CONCAT('DUP_INT_', F_CodeToHex(aOCVFileCodeName[1]));
		stOCVStatus.nStatus.22 := TRUE;

		bDuplicateInterimFound := TRUE;
END_IF
END_ACTION

ACTION DuplicatePackFound:
FOR nPackCodeCheckIndex:= 1 TO nPacksPerOuter DO
	FOR nPackCodeDupIndex := 1 TO nPacksPerOuter DO

		IF  stNextOCVStatus.nStatus.6
			AND stOCVStatus.stOACData.PackCode[nPackCodeCheckIndex] = stNextOCVStatus.stOACData.PackCode[nPackCodeDupIndex]
			AND (stOCVStatus.aOACPackStatus[nPackCodeCheckIndex] = 5 OR  stOCVStatus.aOACPackStatus[nPackCodeCheckIndex] = 6) THEN

				aOCVFileCodeToDelete[1]	:=	F_CodeToHex(F_CODE_GetItem(stNextOCVStatus.stOACData.AggregationCodes[1] ,
																eCodeAIType.SerialCode, SEL(bUseIntermediateCode, stCodeInfo_Pack, stCodeInfo_Intermediate)));
				aOCVFileCodeToDelete[2]	:=	F_CodeToHex(F_CODE_GetItem(stNextOCVStatus.stOACData.AggregationCodes[2] ,
																eCodeAIType.SerialCode, stCodeInfo_Pack));

				stNextOCVStatus.nStatus.22 := TRUE;
				stNextOCVStatus.sDataSourceTracker  := 'REMOVED';

				aOCVFileCodeName[1] := F_CONCAT5('DUP_PK1_', F_CodeToHex(aOCVFileCodeName[1]),'_' , F_SYSTEM_SystemTimeToCHM_Header(stCTDateTime.sSystemTime), '.xml');
				aOCVFileCodeName[2] := F_CONCAT5('DUP_PK2_', F_CodeToHex(aOCVFileCodeName[2]),'_' , F_SYSTEM_SystemTimeToCHM_Header(stCTDateTime.sSystemTime), '.xml');
				stOCVStatus.nStatus.22 := TRUE;
				stOCVStatus.sDataSourceTracker  := 'DUPLICAT';

			bDuplicatePackFound := TRUE;
			EXIT;
		END_IF
	END_FOR
	IF bDuplicatePackFound THEN
		EXIT;
	END_IF
END_FOR
END_ACTION

ACTION InvalidPackFound:
FOR nPackCodeCheckIndex := 1 TO nPacksPerOuter DO
	IF stOCVStatus.aOACPackStatus[nPackCodeCheckIndex] = 0
		OR stOCVStatus.aOACPackStatus[nPackCodeCheckIndex] = 1
		OR stOCVStatus.aOACPackStatus[nPackCodeCheckIndex] = 2
		OR stOCVStatus.aOACPackStatus[nPackCodeCheckIndex] = 3	THEN

		bInvalidPackFound := TRUE;
		EXIT;
	END_IF
END_FOR
END_ACTION

ACTION MasterListFound:
FOR nPackCodeCheckIndex := 1 TO nPacksPerOuter DO
	IF stOCVStatus.aOACPackStatus[nPackCodeCheckIndex] = 6 THEN

		aOCVFileCodeName[1] := CONCAT('ML_', F_CodeToHex(aOCVFileCodeName[1]));
		aOCVFileCodeName[2] := CONCAT('ML_', F_CodeToHex(aOCVFileCodeName[2]));

		bMasterListFound	:= TRUE;
		EXIT;
	END_IF
END_FOR
END_ACTION

END_FUNCTION_BLOCK

